//     PlcTask Inputs/GVL_iXlinker.EtherCAT_Master_EPPxxxx.Beckhoff_EPP1xxx.Beckhoff_EPP1xxxEK1122.A_0018_EPP1321_0060_0016.A_0019_EPP1322_0001_0016.A_0020_EPP1322_0001_0017.A_0021_EPP1332_0001_0016.A_0022_EPP1332_0001_0017.A_0023_EPP1342_0001_0016.A_0024_EPP1342_0001_0017.A_0027_EPP1809_0021_0016.WcState.WcState <-> WcState/WcState
//     PlcTask Inputs/GVL_iXlinker.EtherCAT_Master_EPPxxxx.Beckhoff_EPP1xxx.Beckhoff_EPP1xxxEK1122.A_0018_EPP1321_0060_0016.A_0019_EPP1322_0001_0016.A_0020_EPP1322_0001_0017.A_0021_EPP1332_0001_0016.A_0022_EPP1332_0001_0017.A_0023_EPP1342_0001_0016.A_0024_EPP1342_0001_0017.A_0027_EPP1809_0021_0016.WcState.InputToggle <-> WcState/InputToggle
//     PlcTask Inputs/GVL_iXlinker.EtherCAT_Master_EPPxxxx.Beckhoff_EPP1xxx.Beckhoff_EPP1xxxEK1122.A_0018_EPP1321_0060_0016.A_0019_EPP1322_0001_0016.A_0020_EPP1322_0001_0017.A_0021_EPP1332_0001_0016.A_0022_EPP1332_0001_0017.A_0023_EPP1342_0001_0016.A_0024_EPP1342_0001_0017.A_0027_EPP1809_0021_0016.InfoData.State <-> InfoData/State
//   PLC/PLC Instance <-> EtherCAT Master EPPxxxx/Beckhoff EPP1xxx/Beckhoff EPP1xxxEK1122/A_0018(EPP1321-0060-0016)/A_0019(EPP1322-0001-0016)/A_0020(EPP1322-0001-0017)/A_0021(EPP1332-0001-0016)/A_0022(EPP1332-0001-0017)/A_0023(EPP1342-0001-0016)/A_0024(EPP1342-0001-0017)/A_0028(EPP1809-0022-0016)
//     PlcTask Inputs/GVL_iXlinker.EtherCAT_Master_EPPxxxx.Beckhoff_EPP1xxx.Beckhoff_EPP1xxxEK1122.A_0018_EPP1321_0060_0016.A_0019_EPP1322_0001_0016.A_0020_EPP1322_0001_0017.A_0021_EPP1332_0001_0016.A_0022_EPP1332_0001_0017.A_0023_EPP1342_0001_0016.A_0024_EPP1342_0001_0017.A_0028_EPP1809_0022_0016.Channel_1.Input <-> Channel 1/Input
//     PlcTask Inputs/GVL_iXlinker.EtherCAT_Master_EPPxxxx.Beckhoff_EPP1xxx.Beckhoff_EPP1xxxEK1122.A_0018_EPP1321_0060_0016.A_0019_EPP1322_0001_0016.A_0020_EPP1322_0001_0017.A_0021_EPP1332_0001_0016.A_0022_EPP1332_0001_0017.A_0023_EPP1342_0001_0016.A_0024_EPP1342_0001_0017.A_0028_EPP1809_0022_0016.Channel_2.Input <-> Channel 2/Input
//     PlcTask Inputs/GVL_iXlinker.EtherCAT_Master_EPPxxxx.Beckhoff_EPP1xxx.Beckhoff_EPP1xxxEK1122.A_0018_EPP1321_0060_0016.A_0019_EPP1322_0001_0016.A_0020_EPP1322_0001_0017.A_0021_EPP1332_0001_0016.A_0022_EPP1332_0001_0017.A_0023_EPP1342_0001_0016.A_0024_EPP1342_0001_0017.A_0028_EPP1809_0022_0016.Channel_3.Input <-> Channel 3/Input
//     PlcTask Inputs/GVL_iXlinker.EtherCAT_Master_EPPxxxx.Beckhoff_EPP1xxx.Beckhoff_EPP1xxxEK1122.A_0018_EPP1321_0060_0016.A_0019_EPP1322_0001_0016.A_0020_EPP1322_0001_0017.A_0021_EPP1332_0001_0016.A_0022_EPP1332_0001_0017.A_0023_EPP1342_0001_0016.A_0024_EPP1342_0001_0017.A_0028_EPP1809_0022_0016.Channel_4.Input <-> Channel 4/Input
//     PlcTask Inputs/GVL_iXlinker.EtherCAT_Master_EPPxxxx.Beckhoff_EPP1xxx.Beckhoff_EPP1xxxEK1122.A_0018_EPP1321_0060_0016.A_0019_EPP1322_0001_0016.A_0020_EPP1322_0001_0017.A_0021_EPP1332_0001_0016.A_0022_EPP1332_0001_0017.A_0023_EPP1342_0001_0016.A_0024_EPP1342_0001_0017.A_0028_EPP1809_0022_0016.Channel_5.Input <-> Channel 5/Input
//     PlcTask Inputs/GVL_iXlinker.EtherCAT_Master_EPPxxxx.Beckhoff_EPP1xxx.Beckhoff_EPP1xxxEK1122.A_0018_EPP1321_0060_0016.A_0019_EPP1322_0001_0016.A_0020_EPP1322_0001_0017.A_0021_EPP1332_0001_0016.A_0022_EPP1332_0001_0017.A_0023_EPP1342_0001_0016.A_0024_EPP1342_0001_0017.A_0028_EPP1809_0022_0016.Channel_6.Input <-> Channel 6/Input
//     PlcTask Inputs/GVL_iXlinker.EtherCAT_Master_EPPxxxx.Beckhoff_EPP1xxx.Beckhoff_EPP1xxxEK1122.A_0018_EPP1321_0060_0016.A_0019_EPP1322_0001_0016.A_0020_EPP1322_0001_0017.A_0021_EPP1332_0001_0016.A_0022_EPP1332_0001_0017.A_0023_EPP1342_0001_0016.A_0024_EPP1342_0001_0017.A_0028_EPP1809_0022_0016.Channel_7.Input <-> Channel 7/Input
//     PlcTask Inputs/GVL_iXlinker.EtherCAT_Master_EPPxxxx.Beckhoff_EPP1xxx.Beckhoff_EPP1xxxEK1122.A_0018_EPP1321_0060_0016.A_0019_EPP1322_0001_0016.A_0020_EPP1322_0001_0017.A_0021_EPP1332_0001_0016.A_0022_EPP1332_0001_0017.A_0023_EPP1342_0001_0016.A_0024_EPP1342_0001_0017.A_0028_EPP1809_0022_0016.Channel_8.Input <-> Channel 8/Input
//     PlcTask Inputs/GVL_iXlinker.EtherCAT_Master_EPPxxxx.Beckhoff_EPP1xxx.Beckhoff_EPP1xxxEK1122.A_0018_EPP1321_0060_0016.A_0019_EPP1322_0001_0016.A_0020_EPP1322_0001_0017.A_0021_EPP1332_0001_0016.A_0022_EPP1332_0001_0017.A_0023_EPP1342_0001_0016.A_0024_EPP1342_0001_0017.A_0028_EPP1809_0022_0016.Channel_9.Input <-> Channel 9/Input
//     PlcTask Inputs/GVL_iXlinker.EtherCAT_Master_EPPxxxx.Beckhoff_EPP1xxx.Beckhoff_EPP1xxxEK1122.A_0018_EPP1321_0060_0016.A_0019_EPP1322_0001_0016.A_0020_EPP1322_0001_0017.A_0021_EPP1332_0001_0016.A_0022_EPP1332_0001_0017.A_0023_EPP1342_0001_0016.A_0024_EPP1342_0001_0017.A_0028_EPP1809_0022_0016.Channel_10.Input <-> Channel 10/Input
//     PlcTask Inputs/GVL_iXlinker.EtherCAT_Master_EPPxxxx.Beckhoff_EPP1xxx.Beckhoff_EPP1xxxEK1122.A_0018_EPP1321_0060_0016.A_0019_EPP1322_0001_0016.A_0020_EPP1322_0001_0017.A_0021_EPP1332_0001_0016.A_0022_EPP1332_0001_0017.A_0023_EPP1342_0001_0016.A_0024_EPP1342_0001_0017.A_0028_EPP1809_0022_0016.Channel_11.Input <-> Channel 11/Input
//     PlcTask Inputs/GVL_iXlinker.EtherCAT_Master_EPPxxxx.Beckhoff_EPP1xxx.Beckhoff_EPP1xxxEK1122.A_0018_EPP1321_0060_0016.A_0019_EPP1322_0001_0016.A_0020_EPP1322_0001_0017.A_0021_EPP1332_0001_0016.A_0022_EPP1332_0001_0017.A_0023_EPP1342_0001_0016.A_0024_EPP1342_0001_0017.A_0028_EPP1809_0022_0016.Channel_12.Input <-> Channel 12/Input
//     PlcTask Inputs/GVL_iXlinker.EtherCAT_Master_EPPxxxx.Beckhoff_EPP1xxx.Beckhoff_EPP1xxxEK1122.A_0018_EPP1321_0060_0016.A_0019_EPP1322_0001_0016.A_0020_EPP1322_0001_0017.A_0021_EPP1332_0001_0016.A_0022_EPP1332_0001_0017.A_0023_EPP1342_0001_0016.A_0024_EPP1342_0001_0017.A_0028_EPP1809_0022_0016.Channel_13.Input <-> Channel 13/Input
//     PlcTask Inputs/GVL_iXlinker.EtherCAT_Master_EPPxxxx.Beckhoff_EPP1xxx.Beckhoff_EPP1xxxEK1122.A_0018_EPP1321_0060_0016.A_0019_EPP1322_0001_0016.A_0020_EPP1322_0001_0017.A_0021_EPP1332_0001_0016.A_0022_EPP1332_0001_0017.A_0023_EPP1342_0001_0016.A_0024_EPP1342_0001_0017.A_0028_EPP1809_0022_0016.Channel_14.Input <-> Channel 14/Input
//     PlcTask Inputs/GVL_iXlinker.EtherCAT_Master_EPPxxxx.Beckhoff_EPP1xxx.Beckhoff_EPP1xxxEK1122.A_0018_EPP1321_0060_0016.A_0019_EPP1322_0001_0016.A_0020_EPP1322_0001_0017.A_0021_EPP1332_0001_0016.A_0022_EPP1332_0001_0017.A_0023_EPP1342_0001_0016.A_0024_EPP1342_0001_0017.A_0028_EPP1809_0022_0016.Channel_15.Input <-> Channel 15/Input
//     PlcTask Inputs/GVL_iXlinker.EtherCAT_Master_EPPxxxx.Beckhoff_EPP1xxx.Beckhoff_EPP1xxxEK1122.A_0018_EPP1321_0060_0016.A_0019_EPP1322_0001_0016.A_0020_EPP1322_0001_0017.A_0021_EPP1332_0001_0016.A_0022_EPP1332_0001_0017.A_0023_EPP1342_0001_0016.A_0024_EPP1342_0001_0017.A_0028_EPP1809_0022_0016.Channel_16.Input <-> Channel 16/Input
//     PlcTask Inputs/GVL_iXlinker.EtherCAT_Master_EPPxxxx.Beckhoff_EPP1xxx.Beckhoff_EPP1xxxEK1122.A_0018_EPP1321_0060_0016.A_0019_EPP1322_0001_0016.A_0020_EPP1322_0001_0017.A_0021_EPP1332_0001_0016.A_0022_EPP1332_0001_0017.A_0023_EPP1342_0001_0016.A_0024_EPP1342_0001_0017.A_0028_EPP1809_0022_0016.WcState.WcState <-> WcState/WcState
//     PlcTask Inputs/GVL_iXlinker.EtherCAT_Master_EPPxxxx.Beckhoff_EPP1xxx.Beckhoff_EPP1xxxEK1122.A_0018_EPP1321_0060_0016.A_0019_EPP1322_0001_0016.A_0020_EPP1322_0001_0017.A_0021_EPP1332_0001_0016.A_0022_EPP1332_0001_0017.A_0023_EPP1342_0001_0016.A_0024_EPP1342_0001_0017.A_0028_EPP1809_0022_0016.WcState.InputToggle <-> WcState/InputToggle
//     PlcTask Inputs/GVL_iXlinker.EtherCAT_Master_EPPxxxx.Beckhoff_EPP1xxx.Beckhoff_EPP1xxxEK1122.A_0018_EPP1321_0060_0016.A_0019_EPP1322_0001_0016.A_0020_EPP1322_0001_0017.A_0021_EPP1332_0001_0016.A_0022_EPP1332_0001_0017.A_0023_EPP1342_0001_0016.A_0024_EPP1342_0001_0017.A_0028_EPP1809_0022_0016.InfoData.State <-> InfoData/State
//   PLC/PLC Instance <-> EtherCAT Master EPPxxxx/Beckhoff EPP1xxx/Beckhoff EPP1xxxEK1122/A_0018(EPP1321-0060-0016)/A_0019(EPP1322-0001-0016)/A_0020(EPP1322-0001-0017)/A_0021(EPP1332-0001-0016)/A_0022(EPP1332-0001-0017)/A_0023(EPP1342-0001-0016)/A_0024(EPP1342-0001-0017)/A_0029(EPP1819-0021-0016)
//     PlcTask Inputs/GVL_iXlinker.EtherCAT_Master_EPPxxxx.Beckhoff_EPP1xxx.Beckhoff_EPP1xxxEK1122.A_0018_EPP1321_0060_0016.A_0019_EPP1322_0001_0016.A_0020_EPP1322_0001_0017.A_0021_EPP1332_0001_0016.A_0022_EPP1332_0001_0017.A_0023_EPP1342_0001_0016.A_0024_EPP1342_0001_0017.A_0029_EPP1819_0021_0016.Channel_1.Input <-> Channel 1/Input
//     PlcTask Inputs/GVL_iXlinker.EtherCAT_Master_EPPxxxx.Beckhoff_EPP1xxx.Beckhoff_EPP1xxxEK1122.A_0018_EPP1321_0060_0016.A_0019_EPP1322_0001_0016.A_0020_EPP1322_0001_0017.A_0021_EPP1332_0001_0016.A_0022_EPP1332_0001_0017.A_0023_EPP1342_0001_0016.A_0024_EPP1342_0001_0017.A_0029_EPP1819_0021_0016.Channel_2.Input <-> Channel 2/Input
//     PlcTask Inputs/GVL_iXlinker.EtherCAT_Master_EPPxxxx.Beckhoff_EPP1xxx.Beckhoff_EPP1xxxEK1122.A_0018_EPP1321_0060_0016.A_0019_EPP1322_0001_0016.A_0020_EPP1322_0001_0017.A_0021_EPP1332_0001_0016.A_0022_EPP1332_0001_0017.A_0023_EPP1342_0001_0016.A_0024_EPP1342_0001_0017.A_0029_EPP1819_0021_0016.Channel_3.Input <-> Channel 3/Input
//     PlcTask Inputs/GVL_iXlinker.EtherCAT_Master_EPPxxxx.Beckhoff_EPP1xxx.Beckhoff_EPP1xxxEK1122.A_0018_EPP1321_0060_0016.A_0019_EPP1322_0001_0016.A_0020_EPP1322_0001_0017.A_0021_EPP1332_0001_0016.A_0022_EPP1332_0001_0017.A_0023_EPP1342_0001_0016.A_0024_EPP1342_0001_0017.A_0029_EPP1819_0021_0016.Channel_4.Input <-> Channel 4/Input
//     PlcTask Inputs/GVL_iXlinker.EtherCAT_Master_EPPxxxx.Beckhoff_EPP1xxx.Beckhoff_EPP1xxxEK1122.A_0018_EPP1321_0060_0016.A_0019_EPP1322_0001_0016.A_0020_EPP1322_0001_0017.A_0021_EPP1332_0001_0016.A_0022_EPP1332_0001_0017.A_0023_EPP1342_0001_0016.A_0024_EPP1342_0001_0017.A_0029_EPP1819_0021_0016.Channel_5.Input <-> Channel 5/Input
//     PlcTask Inputs/GVL_iXlinker.EtherCAT_Master_EPPxxxx.Beckhoff_EPP1xxx.Beckhoff_EPP1xxxEK1122.A_0018_EPP1321_0060_0016.A_0019_EPP1322_0001_0016.A_0020_EPP1322_0001_0017.A_0021_EPP1332_0001_0016.A_0022_EPP1332_0001_0017.A_0023_EPP1342_0001_0016.A_0024_EPP1342_0001_0017.A_0029_EPP1819_0021_0016.Channel_6.Input <-> Channel 6/Input
//     PlcTask Inputs/GVL_iXlinker.EtherCAT_Master_EPPxxxx.Beckhoff_EPP1xxx.Beckhoff_EPP1xxxEK1122.A_0018_EPP1321_0060_0016.A_0019_EPP1322_0001_0016.A_0020_EPP1322_0001_0017.A_0021_EPP1332_0001_0016.A_0022_EPP1332_0001_0017.A_0023_EPP1342_0001_0016.A_0024_EPP1342_0001_0017.A_0029_EPP1819_0021_0016.Channel_7.Input <-> Channel 7/Input
//     PlcTask Inputs/GVL_iXlinker.EtherCAT_Master_EPPxxxx.Beckhoff_EPP1xxx.Beckhoff_EPP1xxxEK1122.A_0018_EPP1321_0060_0016.A_0019_EPP1322_0001_0016.A_0020_EPP1322_0001_0017.A_0021_EPP1332_0001_0016.A_0022_EPP1332_0001_0017.A_0023_EPP1342_0001_0016.A_0024_EPP1342_0001_0017.A_0029_EPP1819_0021_0016.Channel_8.Input <-> Channel 8/Input
//     PlcTask Inputs/GVL_iXlinker.EtherCAT_Master_EPPxxxx.Beckhoff_EPP1xxx.Beckhoff_EPP1xxxEK1122.A_0018_EPP1321_0060_0016.A_0019_EPP1322_0001_0016.A_0020_EPP1322_0001_0017.A_0021_EPP1332_0001_0016.A_0022_EPP1332_0001_0017.A_0023_EPP1342_0001_0016.A_0024_EPP1342_0001_0017.A_0029_EPP1819_0021_0016.Channel_9.Input <-> Channel 9/Input
//     PlcTask Inputs/GVL_iXlinker.EtherCAT_Master_EPPxxxx.Beckhoff_EPP1xxx.Beckhoff_EPP1xxxEK1122.A_0018_EPP1321_0060_0016.A_0019_EPP1322_0001_0016.A_0020_EPP1322_0001_0017.A_0021_EPP1332_0001_0016.A_0022_EPP1332_0001_0017.A_0023_EPP1342_0001_0016.A_0024_EPP1342_0001_0017.A_0029_EPP1819_0021_0016.Channel_10.Input <-> Channel 10/Input
//     PlcTask Inputs/GVL_iXlinker.EtherCAT_Master_EPPxxxx.Beckhoff_EPP1xxx.Beckhoff_EPP1xxxEK1122.A_0018_EPP1321_0060_0016.A_0019_EPP1322_0001_0016.A_0020_EPP1322_0001_0017.A_0021_EPP1332_0001_0016.A_0022_EPP1332_0001_0017.A_0023_EPP1342_0001_0016.A_0024_EPP1342_0001_0017.A_0029_EPP1819_0021_0016.Channel_11.Input <-> Channel 11/Input
//     PlcTask Inputs/GVL_iXlinker.EtherCAT_Master_EPPxxxx.Beckhoff_EPP1xxx.Beckhoff_EPP1xxxEK1122.A_0018_EPP1321_0060_0016.A_0019_EPP1322_0001_0016.A_0020_EPP1322_0001_0017.A_0021_EPP1332_0001_0016.A_0022_EPP1332_0001_0017.A_0023_EPP1342_0001_0016.A_0024_EPP1342_0001_0017.A_0029_EPP1819_0021_0016.Channel_12.Input <-> Channel 12/Input
//     PlcTask Inputs/GVL_iXlinker.EtherCAT_Master_EPPxxxx.Beckhoff_EPP1xxx.Beckhoff_EPP1xxxEK1122.A_0018_EPP1321_0060_0016.A_0019_EPP1322_0001_0016.A_0020_EPP1322_0001_0017.A_0021_EPP1332_0001_0016.A_0022_EPP1332_0001_0017.A_0023_EPP1342_0001_0016.A_0024_EPP1342_0001_0017.A_0029_EPP1819_0021_0016.Channel_13.Input <-> Channel 13/Input
//     PlcTask Inputs/GVL_iXlinker.EtherCAT_Master_EPPxxxx.Beckhoff_EPP1xxx.Beckhoff_EPP1xxxEK1122.A_0018_EPP1321_0060_0016.A_0019_EPP1322_0001_0016.A_0020_EPP1322_0001_0017.A_0021_EPP1332_0001_0016.A_0022_EPP1332_0001_0017.A_0023_EPP1342_0001_0016.A_0024_EPP1342_0001_0017.A_0029_EPP1819_0021_0016.Channel_14.Input <-> Channel 14/Input
//     PlcTask Inputs/GVL_iXlinker.EtherCAT_Master_EPPxxxx.Beckhoff_EPP1xxx.Beckhoff_EPP1xxxEK1122.A_0018_EPP1321_0060_0016.A_0019_EPP1322_0001_0016.A_0020_EPP1322_0001_0017.A_0021_EPP1332_0001_0016.A_0022_EPP1332_0001_0017.A_0023_EPP1342_0001_0016.A_0024_EPP1342_0001_0017.A_0029_EPP1819_0021_0016.Channel_15.Input <-> Channel 15/Input
//     PlcTask Inputs/GVL_iXlinker.EtherCAT_Master_EPPxxxx.Beckhoff_EPP1xxx.Beckhoff_EPP1xxxEK1122.A_0018_EPP1321_0060_0016.A_0019_EPP1322_0001_0016.A_0020_EPP1322_0001_0017.A_0021_EPP1332_0001_0016.A_0022_EPP1332_0001_0017.A_0023_EPP1342_0001_0016.A_0024_EPP1342_0001_0017.A_0029_EPP1819_0021_0016.Channel_16.Input <-> Channel 16/Input
//     PlcTask Inputs/GVL_iXlinker.EtherCAT_Master_EPPxxxx.Beckhoff_EPP1xxx.Beckhoff_EPP1xxxEK1122.A_0018_EPP1321_0060_0016.A_0019_EPP1322_0001_0016.A_0020_EPP1322_0001_0017.A_0021_EPP1332_0001_0016.A_0022_EPP1332_0001_0017.A_0023_EPP1342_0001_0016.A_0024_EPP1342_0001_0017.A_0029_EPP1819_0021_0016.WcState.WcState <-> WcState/WcState
//     PlcTask Inputs/GVL_iXlinker.EtherCAT_Master_EPPxxxx.Beckhoff_EPP1xxx.Beckhoff_EPP1xxxEK1122.A_0018_EPP1321_0060_0016.A_0019_EPP1322_0001_0016.A_0020_EPP1322_0001_0017.A_0021_EPP1332_0001_0016.A_0022_EPP1332_0001_0017.A_0023_EPP1342_0001_0016.A_0024_EPP1342_0001_0017.A_0029_EPP1819_0021_0016.WcState.InputToggle <-> WcState/InputToggle
//     PlcTask Inputs/GVL_iXlinker.EtherCAT_Master_EPPxxxx.Beckhoff_EPP1xxx.Beckhoff_EPP1xxxEK1122.A_0018_EPP1321_0060_0016.A_0019_EPP1322_0001_0016.A_0020_EPP1322_0001_0017.A_0021_EPP1332_0001_0016.A_0022_EPP1332_0001_0017.A_0023_EPP1342_0001_0016.A_0024_EPP1342_0001_0017.A_0029_EPP1819_0021_0016.InfoData.State <-> InfoData/State
//   PLC/PLC Instance <-> EtherCAT Master EPPxxxx/Beckhoff EPP1xxx/Beckhoff EPP1xxxEK1122/A_0018(EPP1321-0060-0016)/A_0019(EPP1322-0001-0016)/A_0020(EPP1322-0001-0017)/A_0021(EPP1332-0001-0016)/A_0022(EPP1332-0001-0017)/A_0023(EPP1342-0001-0016)/A_0024(EPP1342-0001-0017)/A_0030(EPP1819-0022-0016)
//     PlcTask Inputs/GVL_iXlinker.EtherCAT_Master_EPPxxxx.Beckhoff_EPP1xxx.Beckhoff_EPP1xxxEK1122.A_0018_EPP1321_0060_0016.A_0019_EPP1322_0001_0016.A_0020_EPP1322_0001_0017.A_0021_EPP1332_0001_0016.A_0022_EPP1332_0001_0017.A_0023_EPP1342_0001_0016.A_0024_EPP1342_0001_0017.A_0030_EPP1819_0022_0016.Channel_1.Input <-> Channel 1/Input
//     PlcTask Inputs/GVL_iXlinker.EtherCAT_Master_EPPxxxx.Beckhoff_EPP1xxx.Beckhoff_EPP1xxxEK1122.A_0018_EPP1321_0060_0016.A_0019_EPP1322_0001_0016.A_0020_EPP1322_0001_0017.A_0021_EPP1332_0001_0016.A_0022_EPP1332_0001_0017.A_0023_EPP1342_0001_0016.A_0024_EPP1342_0001_0017.A_0030_EPP1819_0022_0016.Channel_2.Input <-> Channel 2/Input
//     PlcTask Inputs/GVL_iXlinker.EtherCAT_Master_EPPxxxx.Beckhoff_EPP1xxx.Beckhoff_EPP1xxxEK1122.A_0018_EPP1321_0060_0016.A_0019_EPP1322_0001_0016.A_0020_EPP1322_0001_0017.A_0021_EPP1332_0001_0016.A_0022_EPP1332_0001_0017.A_0023_EPP1342_0001_0016.A_0024_EPP1342_0001_0017.A_0030_EPP1819_0022_0016.Channel_3.Input <-> Channel 3/Input
//     PlcTask Inputs/GVL_iXlinker.EtherCAT_Master_EPPxxxx.Beckhoff_EPP1xxx.Beckhoff_EPP1xxxEK1122.A_0018_EPP1321_0060_0016.A_0019_EPP1322_0001_0016.A_0020_EPP1322_0001_0017.A_0021_EPP1332_0001_0016.A_0022_EPP1332_0001_0017.A_0023_EPP1342_0001_0016.A_0024_EPP1342_0001_0017.A_0030_EPP1819_0022_0016.Channel_4.Input <-> Channel 4/Input
//     PlcTask Inputs/GVL_iXlinker.EtherCAT_Master_EPPxxxx.Beckhoff_EPP1xxx.Beckhoff_EPP1xxxEK1122.A_0018_EPP1321_0060_0016.A_0019_EPP1322_0001_0016.A_0020_EPP1322_0001_0017.A_0021_EPP1332_0001_0016.A_0022_EPP1332_0001_0017.A_0023_EPP1342_0001_0016.A_0024_EPP1342_0001_0017.A_0030_EPP1819_0022_0016.Channel_5.Input <-> Channel 5/Input
//     PlcTask Inputs/GVL_iXlinker.EtherCAT_Master_EPPxxxx.Beckhoff_EPP1xxx.Beckhoff_EPP1xxxEK1122.A_0018_EPP1321_0060_0016.A_0019_EPP1322_0001_0016.A_0020_EPP1322_0001_0017.A_0021_EPP1332_0001_0016.A_0022_EPP1332_0001_0017.A_0023_EPP1342_0001_0016.A_0024_EPP1342_0001_0017.A_0030_EPP1819_0022_0016.Channel_6.Input <-> Channel 6/Input
//     PlcTask Inputs/GVL_iXlinker.EtherCAT_Master_EPPxxxx.Beckhoff_EPP1xxx.Beckhoff_EPP1xxxEK1122.A_0018_EPP1321_0060_0016.A_0019_EPP1322_0001_0016.A_0020_EPP1322_0001_0017.A_0021_EPP1332_0001_0016.A_0022_EPP1332_0001_0017.A_0023_EPP1342_0001_0016.A_0024_EPP1342_0001_0017.A_0030_EPP1819_0022_0016.Channel_7.Input <-> Channel 7/Input
//     PlcTask Inputs/GVL_iXlinker.EtherCAT_Master_EPPxxxx.Beckhoff_EPP1xxx.Beckhoff_EPP1xxxEK1122.A_0018_EPP1321_0060_0016.A_0019_EPP1322_0001_0016.A_0020_EPP1322_0001_0017.A_0021_EPP1332_0001_0016.A_0022_EPP1332_0001_0017.A_0023_EPP1342_0001_0016.A_0024_EPP1342_0001_0017.A_0030_EPP1819_0022_0016.Channel_8.Input <-> Channel 8/Input
//     PlcTask Inputs/GVL_iXlinker.EtherCAT_Master_EPPxxxx.Beckhoff_EPP1xxx.Beckhoff_EPP1xxxEK1122.A_0018_EPP1321_0060_0016.A_0019_EPP1322_0001_0016.A_0020_EPP1322_0001_0017.A_0021_EPP1332_0001_0016.A_0022_EPP1332_0001_0017.A_0023_EPP1342_0001_0016.A_0024_EPP1342_0001_0017.A_0030_EPP1819_0022_0016.Channel_9.Input <-> Channel 9/Input
//     PlcTask Inputs/GVL_iXlinker.EtherCAT_Master_EPPxxxx.Beckhoff_EPP1xxx.Beckhoff_EPP1xxxEK1122.A_0018_EPP1321_0060_0016.A_0019_EPP1322_0001_0016.A_0020_EPP1322_0001_0017.A_0021_EPP1332_0001_0016.A_0022_EPP1332_0001_0017.A_0023_EPP1342_0001_0016.A_0024_EPP1342_0001_0017.A_0030_EPP1819_0022_0016.Channel_10.Input <-> Channel 10/Input
//     PlcTask Inputs/GVL_iXlinker.EtherCAT_Master_EPPxxxx.Beckhoff_EPP1xxx.Beckhoff_EPP1xxxEK1122.A_0018_EPP1321_0060_0016.A_0019_EPP1322_0001_0016.A_0020_EPP1322_0001_0017.A_0021_EPP1332_0001_0016.A_0022_EPP1332_0001_0017.A_0023_EPP1342_0001_0016.A_0024_EPP1342_0001_0017.A_0030_EPP1819_0022_0016.Channel_11.Input <-> Channel 11/Input
//     PlcTask Inputs/GVL_iXlinker.EtherCAT_Master_EPPxxxx.Beckhoff_EPP1xxx.Beckhoff_EPP1xxxEK1122.A_0018_EPP1321_0060_0016.A_0019_EPP1322_0001_0016.A_0020_EPP1322_0001_0017.A_0021_EPP1332_0001_0016.A_0022_EPP1332_0001_0017.A_0023_EPP1342_0001_0016.A_0024_EPP1342_0001_0017.A_0030_EPP1819_0022_0016.Channel_12.Input <-> Channel 12/Input
//     PlcTask Inputs/GVL_iXlinker.EtherCAT_Master_EPPxxxx.Beckhoff_EPP1xxx.Beckhoff_EPP1xxxEK1122.A_0018_EPP1321_0060_0016.A_0019_EPP1322_0001_0016.A_0020_EPP1322_0001_0017.A_0021_EPP1332_0001_0016.A_0022_EPP1332_0001_0017.A_0023_EPP1342_0001_0016.A_0024_EPP1342_0001_0017.A_0030_EPP1819_0022_0016.Channel_13.Input <-> Channel 13/Input
//     PlcTask Inputs/GVL_iXlinker.EtherCAT_Master_EPPxxxx.Beckhoff_EPP1xxx.Beckhoff_EPP1xxxEK1122.A_0018_EPP1321_0060_0016.A_0019_EPP1322_0001_0016.A_0020_EPP1322_0001_0017.A_0021_EPP1332_0001_0016.A_0022_EPP1332_0001_0017.A_0023_EPP1342_0001_0016.A_0024_EPP1342_0001_0017.A_0030_EPP1819_0022_0016.Channel_14.Input <-> Channel 14/Input
//     PlcTask Inputs/GVL_iXlinker.EtherCAT_Master_EPPxxxx.Beckhoff_EPP1xxx.Beckhoff_EPP1xxxEK1122.A_0018_EPP1321_0060_0016.A_0019_EPP1322_0001_0016.A_0020_EPP1322_0001_0017.A_0021_EPP1332_0001_0016.A_0022_EPP1332_0001_0017.A_0023_EPP1342_0001_0016.A_0024_EPP1342_0001_0017.A_0030_EPP1819_0022_0016.Channel_15.Input <-> Channel 15/Input
//     PlcTask Inputs/GVL_iXlinker.EtherCAT_Master_EPPxxxx.Beckhoff_EPP1xxx.Beckhoff_EPP1xxxEK1122.A_0018_EPP1321_0060_0016.A_0019_EPP1322_0001_0016.A_0020_EPP1322_0001_0017.A_0021_EPP1332_0001_0016.A_0022_EPP1332_0001_0017.A_0023_EPP1342_0001_0016.A_0024_EPP1342_0001_0017.A_0030_EPP1819_0022_0016.Channel_16.Input <-> Channel 16/Input
//     PlcTask Inputs/GVL_iXlinker.EtherCAT_Master_EPPxxxx.Beckhoff_EPP1xxx.Beckhoff_EPP1xxxEK1122.A_0018_EPP1321_0060_0016.A_0019_EPP1322_0001_0016.A_0020_EPP1322_0001_0017.A_0021_EPP1332_0001_0016.A_0022_EPP1332_0001_0017.A_0023_EPP1342_0001_0016.A_0024_EPP1342_0001_0017.A_0030_EPP1819_0022_0016.WcState.WcState <-> WcState/WcState
//     PlcTask Inputs/GVL_iXlinker.EtherCAT_Master_EPPxxxx.Beckhoff_EPP1xxx.Beckhoff_EPP1xxxEK1122.A_0018_EPP1321_0060_0016.A_0019_EPP1322_0001_0016.A_0020_EPP1322_0001_0017.A_0021_EPP1332_0001_0016.A_0022_EPP1332_0001_0017.A_0023_EPP1342_0001_0016.A_0024_EPP1342_0001_0017.A_0030_EPP1819_0022_0016.WcState.InputToggle <-> WcState/InputToggle
//     PlcTask Inputs/GVL_iXlinker.EtherCAT_Master_EPPxxxx.Beckhoff_EPP1xxx.Beckhoff_EPP1xxxEK1122.A_0018_EPP1321_0060_0016.A_0019_EPP1322_0001_0016.A_0020_EPP1322_0001_0017.A_0021_EPP1332_0001_0016.A_0022_EPP1332_0001_0017.A_0023_EPP1342_0001_0016.A_0024_EPP1342_0001_0017.A_0030_EPP1819_0022_0016.InfoData.State <-> InfoData/State
//   PLC/PLC Instance <-> EtherCAT Master EPPxxxx/Beckhoff EPP1xxx/Beckhoff EPP1xxxEK1122/A_0018(EPP1321-0060-0016)/A_0019(EPP1322-0001-0016)/A_0020(EPP1322-0001-0017)/A_0021(EPP1332-0001-0016)/A_0022(EPP1332-0001-0017)/A_0023(EPP1342-0001-0016)/A_0024(EPP1342-0001-0017)/A_0031(EPP1816-0003-0016)
//     PlcTask Inputs/GVL_iXlinker.EtherCAT_Master_EPPxxxx.Beckhoff_EPP1xxx.Beckhoff_EPP1xxxEK1122.A_0018_EPP1321_0060_0016.A_0019_EPP1322_0001_0016.A_0020_EPP1322_0001_0017.A_0021_EPP1332_0001_0016.A_0022_EPP1332_0001_0017.A_0023_EPP1342_0001_0016.A_0024_EPP1342_0001_0017.A_0031_EPP1816_0003_0016.DIG_Inputs_Channel_1.Input[0] <-> DIG Inputs Channel 1/Input 1
//     PlcTask Inputs/GVL_iXlinker.EtherCAT_Master_EPPxxxx.Beckhoff_EPP1xxx.Beckhoff_EPP1xxxEK1122.A_0018_EPP1321_0060_0016.A_0019_EPP1322_0001_0016.A_0020_EPP1322_0001_0017.A_0021_EPP1332_0001_0016.A_0022_EPP1332_0001_0017.A_0023_EPP1342_0001_0016.A_0024_EPP1342_0001_0017.A_0031_EPP1816_0003_0016.DIG_Inputs_Channel_1.Input[1] <-> DIG Inputs Channel 1/Input 2
//     PlcTask Inputs/GVL_iXlinker.EtherCAT_Master_EPPxxxx.Beckhoff_EPP1xxx.Beckhoff_EPP1xxxEK1122.A_0018_EPP1321_0060_0016.A_0019_EPP1322_0001_0016.A_0020_EPP1322_0001_0017.A_0021_EPP1332_0001_0016.A_0022_EPP1332_0001_0017.A_0023_EPP1342_0001_0016.A_0024_EPP1342_0001_0017.A_0031_EPP1816_0003_0016.DIG_Inputs_Channel_1.Input[2] <-> DIG Inputs Channel 1/Input 3
//     PlcTask Inputs/GVL_iXlinker.EtherCAT_Master_EPPxxxx.Beckhoff_EPP1xxx.Beckhoff_EPP1xxxEK1122.A_0018_EPP1321_0060_0016.A_0019_EPP1322_0001_0016.A_0020_EPP1322_0001_0017.A_0021_EPP1332_0001_0016.A_0022_EPP1332_0001_0017.A_0023_EPP1342_0001_0016.A_0024_EPP1342_0001_0017.A_0031_EPP1816_0003_0016.DIG_Inputs_Channel_1.Input[3] <-> DIG Inputs Channel 1/Input 4
//     PlcTask Inputs/GVL_iXlinker.EtherCAT_Master_EPPxxxx.Beckhoff_EPP1xxx.Beckhoff_EPP1xxxEK1122.A_0018_EPP1321_0060_0016.A_0019_EPP1322_0001_0016.A_0020_EPP1322_0001_0017.A_0021_EPP1332_0001_0016.A_0022_EPP1332_0001_0017.A_0023_EPP1342_0001_0016.A_0024_EPP1342_0001_0017.A_0031_EPP1816_0003_0016.DIG_Inputs_Channel_1.Input[4] <-> DIG Inputs Channel 1/Input 5
//     PlcTask Inputs/GVL_iXlinker.EtherCAT_Master_EPPxxxx.Beckhoff_EPP1xxx.Beckhoff_EPP1xxxEK1122.A_0018_EPP1321_0060_0016.A_0019_EPP1322_0001_0016.A_0020_EPP1322_0001_0017.A_0021_EPP1332_0001_0016.A_0022_EPP1332_0001_0017.A_0023_EPP1342_0001_0016.A_0024_EPP1342_0001_0017.A_0031_EPP1816_0003_0016.DIG_Inputs_Channel_1.Input[5] <-> DIG Inputs Channel 1/Input 6
//     PlcTask Inputs/GVL_iXlinker.EtherCAT_Master_EPPxxxx.Beckhoff_EPP1xxx.Beckhoff_EPP1xxxEK1122.A_0018_EPP1321_0060_0016.A_0019_EPP1322_0001_0016.A_0020_EPP1322_0001_0017.A_0021_EPP1332_0001_0016.A_0022_EPP1332_0001_0017.A_0023_EPP1342_0001_0016.A_0024_EPP1342_0001_0017.A_0031_EPP1816_0003_0016.DIG_Inputs_Channel_1.Input[6] <-> DIG Inputs Channel 1/Input 7
//     PlcTask Inputs/GVL_iXlinker.EtherCAT_Master_EPPxxxx.Beckhoff_EPP1xxx.Beckhoff_EPP1xxxEK1122.A_0018_EPP1321_0060_0016.A_0019_EPP1322_0001_0016.A_0020_EPP1322_0001_0017.A_0021_EPP1332_0001_0016.A_0022_EPP1332_0001_0017.A_0023_EPP1342_0001_0016.A_0024_EPP1342_0001_0017.A_0031_EPP1816_0003_0016.DIG_Inputs_Channel_1.Input[7] <-> DIG Inputs Channel 1/Input 8
//     PlcTask Inputs/GVL_iXlinker.EtherCAT_Master_EPPxxxx.Beckhoff_EPP1xxx.Beckhoff_EPP1xxxEK1122.A_0018_EPP1321_0060_0016.A_0019_EPP1322_0001_0016.A_0020_EPP1322_0001_0017.A_0021_EPP1332_0001_0016.A_0022_EPP1332_0001_0017.A_0023_EPP1342_0001_0016.A_0024_EPP1342_0001_0017.A_0031_EPP1816_0003_0016.DIG_Inputs_Channel_2.Input[0] <-> DIG Inputs Channel 2/Input 1
//     PlcTask Inputs/GVL_iXlinker.EtherCAT_Master_EPPxxxx.Beckhoff_EPP1xxx.Beckhoff_EPP1xxxEK1122.A_0018_EPP1321_0060_0016.A_0019_EPP1322_0001_0016.A_0020_EPP1322_0001_0017.A_0021_EPP1332_0001_0016.A_0022_EPP1332_0001_0017.A_0023_EPP1342_0001_0016.A_0024_EPP1342_0001_0017.A_0031_EPP1816_0003_0016.DIG_Inputs_Channel_2.Input[1] <-> DIG Inputs Channel 2/Input 2
//     PlcTask Inputs/GVL_iXlinker.EtherCAT_Master_EPPxxxx.Beckhoff_EPP1xxx.Beckhoff_EPP1xxxEK1122.A_0018_EPP1321_0060_0016.A_0019_EPP1322_0001_0016.A_0020_EPP1322_0001_0017.A_0021_EPP1332_0001_0016.A_0022_EPP1332_0001_0017.A_0023_EPP1342_0001_0016.A_0024_EPP1342_0001_0017.A_0031_EPP1816_0003_0016.DIG_Inputs_Channel_2.Input[2] <-> DIG Inputs Channel 2/Input 3
//     PlcTask Inputs/GVL_iXlinker.EtherCAT_Master_EPPxxxx.Beckhoff_EPP1xxx.Beckhoff_EPP1xxxEK1122.A_0018_EPP1321_0060_0016.A_0019_EPP1322_0001_0016.A_0020_EPP1322_0001_0017.A_0021_EPP1332_0001_0016.A_0022_EPP1332_0001_0017.A_0023_EPP1342_0001_0016.A_0024_EPP1342_0001_0017.A_0031_EPP1816_0003_0016.DIG_Inputs_Channel_2.Input[3] <-> DIG Inputs Channel 2/Input 4
//     PlcTask Inputs/GVL_iXlinker.EtherCAT_Master_EPPxxxx.Beckhoff_EPP1xxx.Beckhoff_EPP1xxxEK1122.A_0018_EPP1321_0060_0016.A_0019_EPP1322_0001_0016.A_0020_EPP1322_0001_0017.A_0021_EPP1332_0001_0016.A_0022_EPP1332_0001_0017.A_0023_EPP1342_0001_0016.A_0024_EPP1342_0001_0017.A_0031_EPP1816_0003_0016.DIG_Inputs_Channel_2.Input[4] <-> DIG Inputs Channel 2/Input 5
//     PlcTask Inputs/GVL_iXlinker.EtherCAT_Master_EPPxxxx.Beckhoff_EPP1xxx.Beckhoff_EPP1xxxEK1122.A_0018_EPP1321_0060_0016.A_0019_EPP1322_0001_0016.A_0020_EPP1322_0001_0017.A_0021_EPP1332_0001_0016.A_0022_EPP1332_0001_0017.A_0023_EPP1342_0001_0016.A_0024_EPP1342_0001_0017.A_0031_EPP1816_0003_0016.DIG_Inputs_Channel_2.Input[5] <-> DIG Inputs Channel 2/Input 6
//     PlcTask Inputs/GVL_iXlinker.EtherCAT_Master_EPPxxxx.Beckhoff_EPP1xxx.Beckhoff_EPP1xxxEK1122.A_0018_EPP1321_0060_0016.A_0019_EPP1322_0001_0016.A_0020_EPP1322_0001_0017.A_0021_EPP1332_0001_0016.A_0022_EPP1332_0001_0017.A_0023_EPP1342_0001_0016.A_0024_EPP1342_0001_0017.A_0031_EPP1816_0003_0016.DIG_Inputs_Channel_2.Input[6] <-> DIG Inputs Channel 2/Input 7
//     PlcTask Inputs/GVL_iXlinker.EtherCAT_Master_EPPxxxx.Beckhoff_EPP1xxx.Beckhoff_EPP1xxxEK1122.A_0018_EPP1321_0060_0016.A_0019_EPP1322_0001_0016.A_0020_EPP1322_0001_0017.A_0021_EPP1332_0001_0016.A_0022_EPP1332_0001_0017.A_0023_EPP1342_0001_0016.A_0024_EPP1342_0001_0017.A_0031_EPP1816_0003_0016.DIG_Inputs_Channel_2.Input[7] <-> DIG Inputs Channel 2/Input 8
//     PlcTask Inputs/GVL_iXlinker.EtherCAT_Master_EPPxxxx.Beckhoff_EPP1xxx.Beckhoff_EPP1xxxEK1122.A_0018_EPP1321_0060_0016.A_0019_EPP1322_0001_0016.A_0020_EPP1322_0001_0017.A_0021_EPP1332_0001_0016.A_0022_EPP1332_0001_0017.A_0023_EPP1342_0001_0016.A_0024_EPP1342_0001_0017.A_0031_EPP1816_0003_0016.DIG_Inputs_Channel_1.Sync_error <-> DIG Inputs Channel 1/Sync error
//     PlcTask Inputs/GVL_iXlinker.EtherCAT_Master_EPPxxxx.Beckhoff_EPP1xxx.Beckhoff_EPP1xxxEK1122.A_0018_EPP1321_0060_0016.A_0019_EPP1322_0001_0016.A_0020_EPP1322_0001_0017.A_0021_EPP1332_0001_0016.A_0022_EPP1332_0001_0017.A_0023_EPP1342_0001_0016.A_0024_EPP1342_0001_0017.A_0031_EPP1816_0003_0016.DIG_Inputs_Channel_2.Sync_error <-> DIG Inputs Channel 2/Sync error
//     PlcTask Inputs/GVL_iXlinker.EtherCAT_Master_EPPxxxx.Beckhoff_EPP1xxx.Beckhoff_EPP1xxxEK1122.A_0018_EPP1321_0060_0016.A_0019_EPP1322_0001_0016.A_0020_EPP1322_0001_0017.A_0021_EPP1332_0001_0016.A_0022_EPP1332_0001_0017.A_0023_EPP1342_0001_0016.A_0024_EPP1342_0001_0017.A_0031_EPP1816_0003_0016.DIG_Inputs_Channel_1.TxPDO_Toggle <-> DIG Inputs Channel 1/TxPDO Toggle
//     PlcTask Inputs/GVL_iXlinker.EtherCAT_Master_EPPxxxx.Beckhoff_EPP1xxx.Beckhoff_EPP1xxxEK1122.A_0018_EPP1321_0060_0016.A_0019_EPP1322_0001_0016.A_0020_EPP1322_0001_0017.A_0021_EPP1332_0001_0016.A_0022_EPP1332_0001_0017.A_0023_EPP1342_0001_0016.A_0024_EPP1342_0001_0017.A_0031_EPP1816_0003_0016.DIG_Inputs_Channel_2.TxPDO_Toggle <-> DIG Inputs Channel 2/TxPDO Toggle
//     PlcTask Inputs/GVL_iXlinker.EtherCAT_Master_EPPxxxx.Beckhoff_EPP1xxx.Beckhoff_EPP1xxxEK1122.A_0018_EPP1321_0060_0016.A_0019_EPP1322_0001_0016.A_0020_EPP1322_0001_0017.A_0021_EPP1332_0001_0016.A_0022_EPP1332_0001_0017.A_0023_EPP1342_0001_0016.A_0024_EPP1342_0001_0017.A_0031_EPP1816_0003_0016.WcState.WcState <-> WcState/WcState
//     PlcTask Inputs/GVL_iXlinker.EtherCAT_Master_EPPxxxx.Beckhoff_EPP1xxx.Beckhoff_EPP1xxxEK1122.A_0018_EPP1321_0060_0016.A_0019_EPP1322_0001_0016.A_0020_EPP1322_0001_0017.A_0021_EPP1332_0001_0016.A_0022_EPP1332_0001_0017.A_0023_EPP1342_0001_0016.A_0024_EPP1342_0001_0017.A_0031_EPP1816_0003_0016.WcState.InputToggle <-> WcState/InputToggle
//     PlcTask Inputs/GVL_iXlinker.EtherCAT_Master_EPPxxxx.Beckhoff_EPP1xxx.Beckhoff_EPP1xxxEK1122.A_0018_EPP1321_0060_0016.A_0019_EPP1322_0001_0016.A_0020_EPP1322_0001_0017.A_0021_EPP1332_0001_0016.A_0022_EPP1332_0001_0017.A_0023_EPP1342_0001_0016.A_0024_EPP1342_0001_0017.A_0031_EPP1816_0003_0016.InfoData.AdsAddr <-> InfoData/AdsAddr
//     PlcTask Inputs/GVL_iXlinker.EtherCAT_Master_EPPxxxx.Beckhoff_EPP1xxx.Beckhoff_EPP1xxxEK1122.A_0018_EPP1321_0060_0016.A_0019_EPP1322_0001_0016.A_0020_EPP1322_0001_0017.A_0021_EPP1332_0001_0016.A_0022_EPP1332_0001_0017.A_0023_EPP1342_0001_0016.A_0024_EPP1342_0001_0017.A_0031_EPP1816_0003_0016.InfoData.State <-> InfoData/State
//   PLC/PLC Instance <-> EtherCAT Master EPPxxxx/Beckhoff EPP1xxx/Beckhoff EPP1xxxEK1122/A_0018(EPP1321-0060-0016)/A_0019(EPP1322-0001-0016)/A_0020(EPP1322-0001-0017)/A_0021(EPP1332-0001-0016)/A_0022(EPP1332-0001-0017)/A_0023(EPP1342-0001-0016)/A_0024(EPP1342-0001-0017)/A_0032(EPP1816-0008-0016)
//     PlcTask Inputs/GVL_iXlinker.EtherCAT_Master_EPPxxxx.Beckhoff_EPP1xxx.Beckhoff_EPP1xxxEK1122.A_0018_EPP1321_0060_0016.A_0019_EPP1322_0001_0016.A_0020_EPP1322_0001_0017.A_0021_EPP1332_0001_0016.A_0022_EPP1332_0001_0017.A_0023_EPP1342_0001_0016.A_0024_EPP1342_0001_0017.A_0032_EPP1816_0008_0016.DIG_Inputs_Channel_1.Input[0] <-> DIG Inputs Channel 1/Input 1
//     PlcTask Inputs/GVL_iXlinker.EtherCAT_Master_EPPxxxx.Beckhoff_EPP1xxx.Beckhoff_EPP1xxxEK1122.A_0018_EPP1321_0060_0016.A_0019_EPP1322_0001_0016.A_0020_EPP1322_0001_0017.A_0021_EPP1332_0001_0016.A_0022_EPP1332_0001_0017.A_0023_EPP1342_0001_0016.A_0024_EPP1342_0001_0017.A_0032_EPP1816_0008_0016.DIG_Inputs_Channel_1.Input[1] <-> DIG Inputs Channel 1/Input 2
//     PlcTask Inputs/GVL_iXlinker.EtherCAT_Master_EPPxxxx.Beckhoff_EPP1xxx.Beckhoff_EPP1xxxEK1122.A_0018_EPP1321_0060_0016.A_0019_EPP1322_0001_0016.A_0020_EPP1322_0001_0017.A_0021_EPP1332_0001_0016.A_0022_EPP1332_0001_0017.A_0023_EPP1342_0001_0016.A_0024_EPP1342_0001_0017.A_0032_EPP1816_0008_0016.DIG_Inputs_Channel_1.Input[2] <-> DIG Inputs Channel 1/Input 3
//     PlcTask Inputs/GVL_iXlinker.EtherCAT_Master_EPPxxxx.Beckhoff_EPP1xxx.Beckhoff_EPP1xxxEK1122.A_0018_EPP1321_0060_0016.A_0019_EPP1322_0001_0016.A_0020_EPP1322_0001_0017.A_0021_EPP1332_0001_0016.A_0022_EPP1332_0001_0017.A_0023_EPP1342_0001_0016.A_0024_EPP1342_0001_0017.A_0032_EPP1816_0008_0016.DIG_Inputs_Channel_1.Input[3] <-> DIG Inputs Channel 1/Input 4
//     PlcTask Inputs/GVL_iXlinker.EtherCAT_Master_EPPxxxx.Beckhoff_EPP1xxx.Beckhoff_EPP1xxxEK1122.A_0018_EPP1321_0060_0016.A_0019_EPP1322_0001_0016.A_0020_EPP1322_0001_0017.A_0021_EPP1332_0001_0016.A_0022_EPP1332_0001_0017.A_0023_EPP1342_0001_0016.A_0024_EPP1342_0001_0017.A_0032_EPP1816_0008_0016.DIG_Inputs_Channel_1.Input[4] <-> DIG Inputs Channel 1/Input 5
//     PlcTask Inputs/GVL_iXlinker.EtherCAT_Master_EPPxxxx.Beckhoff_EPP1xxx.Beckhoff_EPP1xxxEK1122.A_0018_EPP1321_0060_0016.A_0019_EPP1322_0001_0016.A_0020_EPP1322_0001_0017.A_0021_EPP1332_0001_0016.A_0022_EPP1332_0001_0017.A_0023_EPP1342_0001_0016.A_0024_EPP1342_0001_0017.A_0032_EPP1816_0008_0016.DIG_Inputs_Channel_1.Input[5] <-> DIG Inputs Channel 1/Input 6
//     PlcTask Inputs/GVL_iXlinker.EtherCAT_Master_EPPxxxx.Beckhoff_EPP1xxx.Beckhoff_EPP1xxxEK1122.A_0018_EPP1321_0060_0016.A_0019_EPP1322_0001_0016.A_0020_EPP1322_0001_0017.A_0021_EPP1332_0001_0016.A_0022_EPP1332_0001_0017.A_0023_EPP1342_0001_0016.A_0024_EPP1342_0001_0017.A_0032_EPP1816_0008_0016.DIG_Inputs_Channel_1.Input[6] <-> DIG Inputs Channel 1/Input 7
//     PlcTask Inputs/GVL_iXlinker.EtherCAT_Master_EPPxxxx.Beckhoff_EPP1xxx.Beckhoff_EPP1xxxEK1122.A_0018_EPP1321_0060_0016.A_0019_EPP1322_0001_0016.A_0020_EPP1322_0001_0017.A_0021_EPP1332_0001_0016.A_0022_EPP1332_0001_0017.A_0023_EPP1342_0001_0016.A_0024_EPP1342_0001_0017.A_0032_EPP1816_0008_0016.DIG_Inputs_Channel_1.Input[7] <-> DIG Inputs Channel 1/Input 8
//     PlcTask Inputs/GVL_iXlinker.EtherCAT_Master_EPPxxxx.Beckhoff_EPP1xxx.Beckhoff_EPP1xxxEK1122.A_0018_EPP1321_0060_0016.A_0019_EPP1322_0001_0016.A_0020_EPP1322_0001_0017.A_0021_EPP1332_0001_0016.A_0022_EPP1332_0001_0017.A_0023_EPP1342_0001_0016.A_0024_EPP1342_0001_0017.A_0032_EPP1816_0008_0016.DIG_Inputs_Channel_2.Input[0] <-> DIG Inputs Channel 2/Input 1
//     PlcTask Inputs/GVL_iXlinker.EtherCAT_Master_EPPxxxx.Beckhoff_EPP1xxx.Beckhoff_EPP1xxxEK1122.A_0018_EPP1321_0060_0016.A_0019_EPP1322_0001_0016.A_0020_EPP1322_0001_0017.A_0021_EPP1332_0001_0016.A_0022_EPP1332_0001_0017.A_0023_EPP1342_0001_0016.A_0024_EPP1342_0001_0017.A_0032_EPP1816_0008_0016.DIG_Inputs_Channel_2.Input[1] <-> DIG Inputs Channel 2/Input 2
//     PlcTask Inputs/GVL_iXlinker.EtherCAT_Master_EPPxxxx.Beckhoff_EPP1xxx.Beckhoff_EPP1xxxEK1122.A_0018_EPP1321_0060_0016.A_0019_EPP1322_0001_0016.A_0020_EPP1322_0001_0017.A_0021_EPP1332_0001_0016.A_0022_EPP1332_0001_0017.A_0023_EPP1342_0001_0016.A_0024_EPP1342_0001_0017.A_0032_EPP1816_0008_0016.DIG_Inputs_Channel_2.Input[2] <-> DIG Inputs Channel 2/Input 3
//     PlcTask Inputs/GVL_iXlinker.EtherCAT_Master_EPPxxxx.Beckhoff_EPP1xxx.Beckhoff_EPP1xxxEK1122.A_0018_EPP1321_0060_0016.A_0019_EPP1322_0001_0016.A_0020_EPP1322_0001_0017.A_0021_EPP1332_0001_0016.A_0022_EPP1332_0001_0017.A_0023_EPP1342_0001_0016.A_0024_EPP1342_0001_0017.A_0032_EPP1816_0008_0016.DIG_Inputs_Channel_2.Input[3] <-> DIG Inputs Channel 2/Input 4
//     PlcTask Inputs/GVL_iXlinker.EtherCAT_Master_EPPxxxx.Beckhoff_EPP1xxx.Beckhoff_EPP1xxxEK1122.A_0018_EPP1321_0060_0016.A_0019_EPP1322_0001_0016.A_0020_EPP1322_0001_0017.A_0021_EPP1332_0001_0016.A_0022_EPP1332_0001_0017.A_0023_EPP1342_0001_0016.A_0024_EPP1342_0001_0017.A_0032_EPP1816_0008_0016.DIG_Inputs_Channel_2.Input[4] <-> DIG Inputs Channel 2/Input 5
//     PlcTask Inputs/GVL_iXlinker.EtherCAT_Master_EPPxxxx.Beckhoff_EPP1xxx.Beckhoff_EPP1xxxEK1122.A_0018_EPP1321_0060_0016.A_0019_EPP1322_0001_0016.A_0020_EPP1322_0001_0017.A_0021_EPP1332_0001_0016.A_0022_EPP1332_0001_0017.A_0023_EPP1342_0001_0016.A_0024_EPP1342_0001_0017.A_0032_EPP1816_0008_0016.DIG_Inputs_Channel_2.Input[5] <-> DIG Inputs Channel 2/Input 6
//     PlcTask Inputs/GVL_iXlinker.EtherCAT_Master_EPPxxxx.Beckhoff_EPP1xxx.Beckhoff_EPP1xxxEK1122.A_0018_EPP1321_0060_0016.A_0019_EPP1322_0001_0016.A_0020_EPP1322_0001_0017.A_0021_EPP1332_0001_0016.A_0022_EPP1332_0001_0017.A_0023_EPP1342_0001_0016.A_0024_EPP1342_0001_0017.A_0032_EPP1816_0008_0016.DIG_Inputs_Channel_2.Input[6] <-> DIG Inputs Channel 2/Input 7
//     PlcTask Inputs/GVL_iXlinker.EtherCAT_Master_EPPxxxx.Beckhoff_EPP1xxx.Beckhoff_EPP1xxxEK1122.A_0018_EPP1321_0060_0016.A_0019_EPP1322_0001_0016.A_0020_EPP1322_0001_0017.A_0021_EPP1332_0001_0016.A_0022_EPP1332_0001_0017.A_0023_EPP1342_0001_0016.A_0024_EPP1342_0001_0017.A_0032_EPP1816_0008_0016.DIG_Inputs_Channel_2.Input[7] <-> DIG Inputs Channel 2/Input 8
//     PlcTask Inputs/GVL_iXlinker.EtherCAT_Master_EPPxxxx.Beckhoff_EPP1xxx.Beckhoff_EPP1xxxEK1122.A_0018_EPP1321_0060_0016.A_0019_EPP1322_0001_0016.A_0020_EPP1322_0001_0017.A_0021_EPP1332_0001_0016.A_0022_EPP1332_0001_0017.A_0023_EPP1342_0001_0016.A_0024_EPP1342_0001_0017.A_0032_EPP1816_0008_0016.DIG_Inputs_Channel_1.Sync_Error <-> DIG Inputs Channel 1/Sync Error
//     PlcTask Inputs/GVL_iXlinker.EtherCAT_Master_EPPxxxx.Beckhoff_EPP1xxx.Beckhoff_EPP1xxxEK1122.A_0018_EPP1321_0060_0016.A_0019_EPP1322_0001_0016.A_0020_EPP1322_0001_0017.A_0021_EPP1332_0001_0016.A_0022_EPP1332_0001_0017.A_0023_EPP1342_0001_0016.A_0024_EPP1342_0001_0017.A_0032_EPP1816_0008_0016.DIG_Inputs_Channel_2.Sync_Error <-> DIG Inputs Channel 2/Sync Error
//     PlcTask Inputs/GVL_iXlinker.EtherCAT_Master_EPPxxxx.Beckhoff_EPP1xxx.Beckhoff_EPP1xxxEK1122.A_0018_EPP1321_0060_0016.A_0019_EPP1322_0001_0016.A_0020_EPP1322_0001_0017.A_0021_EPP1332_0001_0016.A_0022_EPP1332_0001_0017.A_0023_EPP1342_0001_0016.A_0024_EPP1342_0001_0017.A_0032_EPP1816_0008_0016.WcState.WcState <-> WcState/WcState
//     PlcTask Inputs/GVL_iXlinker.EtherCAT_Master_EPPxxxx.Beckhoff_EPP1xxx.Beckhoff_EPP1xxxEK1122.A_0018_EPP1321_0060_0016.A_0019_EPP1322_0001_0016.A_0020_EPP1322_0001_0017.A_0021_EPP1332_0001_0016.A_0022_EPP1332_0001_0017.A_0023_EPP1342_0001_0016.A_0024_EPP1342_0001_0017.A_0032_EPP1816_0008_0016.WcState.InputToggle <-> WcState/InputToggle
//     PlcTask Inputs/GVL_iXlinker.EtherCAT_Master_EPPxxxx.Beckhoff_EPP1xxx.Beckhoff_EPP1xxxEK1122.A_0018_EPP1321_0060_0016.A_0019_EPP1322_0001_0016.A_0020_EPP1322_0001_0017.A_0021_EPP1332_0001_0016.A_0022_EPP1332_0001_0017.A_0023_EPP1342_0001_0016.A_0024_EPP1342_0001_0017.A_0032_EPP1816_0008_0016.InfoData.AdsAddr <-> InfoData/AdsAddr
//     PlcTask Inputs/GVL_iXlinker.EtherCAT_Master_EPPxxxx.Beckhoff_EPP1xxx.Beckhoff_EPP1xxxEK1122.A_0018_EPP1321_0060_0016.A_0019_EPP1322_0001_0016.A_0020_EPP1322_0001_0017.A_0021_EPP1332_0001_0016.A_0022_EPP1332_0001_0017.A_0023_EPP1342_0001_0016.A_0024_EPP1342_0001_0017.A_0032_EPP1816_0008_0016.InfoData.State <-> InfoData/State
//   PLC/PLC Instance <-> EtherCAT Master EPPxxxx/Beckhoff EPP1xxx/Beckhoff EPP1xxxEK1122/A_0018(EPP1321-0060-0016)/A_0019(EPP1322-0001-0016)/A_0020(EPP1322-0001-0017)/A_0021(EPP1332-0001-0016)/A_0022(EPP1332-0001-0017)/A_0023(EPP1342-0001-0016)/A_0024(EPP1342-0001-0017)/A_0033(EPP1816-0008-0017)
//     PlcTask Inputs/GVL_iXlinker.EtherCAT_Master_EPPxxxx.Beckhoff_EPP1xxx.Beckhoff_EPP1xxxEK1122.A_0018_EPP1321_0060_0016.A_0019_EPP1322_0001_0016.A_0020_EPP1322_0001_0017.A_0021_EPP1332_0001_0016.A_0022_EPP1332_0001_0017.A_0023_EPP1342_0001_0016.A_0024_EPP1342_0001_0017.A_0033_EPP1816_0008_0017.DIG_Inputs_Channel_1.Input[0] <-> DIG Inputs Channel 1/Input 1
//     PlcTask Inputs/GVL_iXlinker.EtherCAT_Master_EPPxxxx.Beckhoff_EPP1xxx.Beckhoff_EPP1xxxEK1122.A_0018_EPP1321_0060_0016.A_0019_EPP1322_0001_0016.A_0020_EPP1322_0001_0017.A_0021_EPP1332_0001_0016.A_0022_EPP1332_0001_0017.A_0023_EPP1342_0001_0016.A_0024_EPP1342_0001_0017.A_0033_EPP1816_0008_0017.DIG_Inputs_Channel_1.Input[1] <-> DIG Inputs Channel 1/Input 2
//     PlcTask Inputs/GVL_iXlinker.EtherCAT_Master_EPPxxxx.Beckhoff_EPP1xxx.Beckhoff_EPP1xxxEK1122.A_0018_EPP1321_0060_0016.A_0019_EPP1322_0001_0016.A_0020_EPP1322_0001_0017.A_0021_EPP1332_0001_0016.A_0022_EPP1332_0001_0017.A_0023_EPP1342_0001_0016.A_0024_EPP1342_0001_0017.A_0033_EPP1816_0008_0017.DIG_Inputs_Channel_1.Input[2] <-> DIG Inputs Channel 1/Input 3
//     PlcTask Inputs/GVL_iXlinker.EtherCAT_Master_EPPxxxx.Beckhoff_EPP1xxx.Beckhoff_EPP1xxxEK1122.A_0018_EPP1321_0060_0016.A_0019_EPP1322_0001_0016.A_0020_EPP1322_0001_0017.A_0021_EPP1332_0001_0016.A_0022_EPP1332_0001_0017.A_0023_EPP1342_0001_0016.A_0024_EPP1342_0001_0017.A_0033_EPP1816_0008_0017.DIG_Inputs_Channel_1.Input[3] <-> DIG Inputs Channel 1/Input 4
//     PlcTask Inputs/GVL_iXlinker.EtherCAT_Master_EPPxxxx.Beckhoff_EPP1xxx.Beckhoff_EPP1xxxEK1122.A_0018_EPP1321_0060_0016.A_0019_EPP1322_0001_0016.A_0020_EPP1322_0001_0017.A_0021_EPP1332_0001_0016.A_0022_EPP1332_0001_0017.A_0023_EPP1342_0001_0016.A_0024_EPP1342_0001_0017.A_0033_EPP1816_0008_0017.DIG_Inputs_Channel_1.Input[4] <-> DIG Inputs Channel 1/Input 5
//     PlcTask Inputs/GVL_iXlinker.EtherCAT_Master_EPPxxxx.Beckhoff_EPP1xxx.Beckhoff_EPP1xxxEK1122.A_0018_EPP1321_0060_0016.A_0019_EPP1322_0001_0016.A_0020_EPP1322_0001_0017.A_0021_EPP1332_0001_0016.A_0022_EPP1332_0001_0017.A_0023_EPP1342_0001_0016.A_0024_EPP1342_0001_0017.A_0033_EPP1816_0008_0017.DIG_Inputs_Channel_1.Input[5] <-> DIG Inputs Channel 1/Input 6
//     PlcTask Inputs/GVL_iXlinker.EtherCAT_Master_EPPxxxx.Beckhoff_EPP1xxx.Beckhoff_EPP1xxxEK1122.A_0018_EPP1321_0060_0016.A_0019_EPP1322_0001_0016.A_0020_EPP1322_0001_0017.A_0021_EPP1332_0001_0016.A_0022_EPP1332_0001_0017.A_0023_EPP1342_0001_0016.A_0024_EPP1342_0001_0017.A_0033_EPP1816_0008_0017.DIG_Inputs_Channel_1.Input[6] <-> DIG Inputs Channel 1/Input 7
//     PlcTask Inputs/GVL_iXlinker.EtherCAT_Master_EPPxxxx.Beckhoff_EPP1xxx.Beckhoff_EPP1xxxEK1122.A_0018_EPP1321_0060_0016.A_0019_EPP1322_0001_0016.A_0020_EPP1322_0001_0017.A_0021_EPP1332_0001_0016.A_0022_EPP1332_0001_0017.A_0023_EPP1342_0001_0016.A_0024_EPP1342_0001_0017.A_0033_EPP1816_0008_0017.DIG_Inputs_Channel_1.Input[7] <-> DIG Inputs Channel 1/Input 8
//     PlcTask Inputs/GVL_iXlinker.EtherCAT_Master_EPPxxxx.Beckhoff_EPP1xxx.Beckhoff_EPP1xxxEK1122.A_0018_EPP1321_0060_0016.A_0019_EPP1322_0001_0016.A_0020_EPP1322_0001_0017.A_0021_EPP1332_0001_0016.A_0022_EPP1332_0001_0017.A_0023_EPP1342_0001_0016.A_0024_EPP1342_0001_0017.A_0033_EPP1816_0008_0017.DIG_Inputs_Channel_2.Input[0] <-> DIG Inputs Channel 2/Input 1
//     PlcTask Inputs/GVL_iXlinker.EtherCAT_Master_EPPxxxx.Beckhoff_EPP1xxx.Beckhoff_EPP1xxxEK1122.A_0018_EPP1321_0060_0016.A_0019_EPP1322_0001_0016.A_0020_EPP1322_0001_0017.A_0021_EPP1332_0001_0016.A_0022_EPP1332_0001_0017.A_0023_EPP1342_0001_0016.A_0024_EPP1342_0001_0017.A_0033_EPP1816_0008_0017.DIG_Inputs_Channel_2.Input[1] <-> DIG Inputs Channel 2/Input 2
//     PlcTask Inputs/GVL_iXlinker.EtherCAT_Master_EPPxxxx.Beckhoff_EPP1xxx.Beckhoff_EPP1xxxEK1122.A_0018_EPP1321_0060_0016.A_0019_EPP1322_0001_0016.A_0020_EPP1322_0001_0017.A_0021_EPP1332_0001_0016.A_0022_EPP1332_0001_0017.A_0023_EPP1342_0001_0016.A_0024_EPP1342_0001_0017.A_0033_EPP1816_0008_0017.DIG_Inputs_Channel_2.Input[2] <-> DIG Inputs Channel 2/Input 3
//     PlcTask Inputs/GVL_iXlinker.EtherCAT_Master_EPPxxxx.Beckhoff_EPP1xxx.Beckhoff_EPP1xxxEK1122.A_0018_EPP1321_0060_0016.A_0019_EPP1322_0001_0016.A_0020_EPP1322_0001_0017.A_0021_EPP1332_0001_0016.A_0022_EPP1332_0001_0017.A_0023_EPP1342_0001_0016.A_0024_EPP1342_0001_0017.A_0033_EPP1816_0008_0017.DIG_Inputs_Channel_2.Input[3] <-> DIG Inputs Channel 2/Input 4
//     PlcTask Inputs/GVL_iXlinker.EtherCAT_Master_EPPxxxx.Beckhoff_EPP1xxx.Beckhoff_EPP1xxxEK1122.A_0018_EPP1321_0060_0016.A_0019_EPP1322_0001_0016.A_0020_EPP1322_0001_0017.A_0021_EPP1332_0001_0016.A_0022_EPP1332_0001_0017.A_0023_EPP1342_0001_0016.A_0024_EPP1342_0001_0017.A_0033_EPP1816_0008_0017.DIG_Inputs_Channel_2.Input[4] <-> DIG Inputs Channel 2/Input 5
//     PlcTask Inputs/GVL_iXlinker.EtherCAT_Master_EPPxxxx.Beckhoff_EPP1xxx.Beckhoff_EPP1xxxEK1122.A_0018_EPP1321_0060_0016.A_0019_EPP1322_0001_0016.A_0020_EPP1322_0001_0017.A_0021_EPP1332_0001_0016.A_0022_EPP1332_0001_0017.A_0023_EPP1342_0001_0016.A_0024_EPP1342_0001_0017.A_0033_EPP1816_0008_0017.DIG_Inputs_Channel_2.Input[5] <-> DIG Inputs Channel 2/Input 6
//     PlcTask Inputs/GVL_iXlinker.EtherCAT_Master_EPPxxxx.Beckhoff_EPP1xxx.Beckhoff_EPP1xxxEK1122.A_0018_EPP1321_0060_0016.A_0019_EPP1322_0001_0016.A_0020_EPP1322_0001_0017.A_0021_EPP1332_0001_0016.A_0022_EPP1332_0001_0017.A_0023_EPP1342_0001_0016.A_0024_EPP1342_0001_0017.A_0033_EPP1816_0008_0017.DIG_Inputs_Channel_2.Input[6] <-> DIG Inputs Channel 2/Input 7
//     PlcTask Inputs/GVL_iXlinker.EtherCAT_Master_EPPxxxx.Beckhoff_EPP1xxx.Beckhoff_EPP1xxxEK1122.A_0018_EPP1321_0060_0016.A_0019_EPP1322_0001_0016.A_0020_EPP1322_0001_0017.A_0021_EPP1332_0001_0016.A_0022_EPP1332_0001_0017.A_0023_EPP1342_0001_0016.A_0024_EPP1342_0001_0017.A_0033_EPP1816_0008_0017.DIG_Inputs_Channel_2.Input[7] <-> DIG Inputs Channel 2/Input 8
//     PlcTask Inputs/GVL_iXlinker.EtherCAT_Master_EPPxxxx.Beckhoff_EPP1xxx.Beckhoff_EPP1xxxEK1122.A_0018_EPP1321_0060_0016.A_0019_EPP1322_0001_0016.A_0020_EPP1322_0001_0017.A_0021_EPP1332_0001_0016.A_0022_EPP1332_0001_0017.A_0023_EPP1342_0001_0016.A_0024_EPP1342_0001_0017.A_0033_EPP1816_0008_0017.DIG_Inputs_Channel_1.Sync_Error <-> DIG Inputs Channel 1/Sync Error
//     PlcTask Inputs/GVL_iXlinker.EtherCAT_Master_EPPxxxx.Beckhoff_EPP1xxx.Beckhoff_EPP1xxxEK1122.A_0018_EPP1321_0060_0016.A_0019_EPP1322_0001_0016.A_0020_EPP1322_0001_0017.A_0021_EPP1332_0001_0016.A_0022_EPP1332_0001_0017.A_0023_EPP1342_0001_0016.A_0024_EPP1342_0001_0017.A_0033_EPP1816_0008_0017.DIG_Inputs_Channel_2.Sync_Error <-> DIG Inputs Channel 2/Sync Error
//     PlcTask Inputs/GVL_iXlinker.EtherCAT_Master_EPPxxxx.Beckhoff_EPP1xxx.Beckhoff_EPP1xxxEK1122.A_0018_EPP1321_0060_0016.A_0019_EPP1322_0001_0016.A_0020_EPP1322_0001_0017.A_0021_EPP1332_0001_0016.A_0022_EPP1332_0001_0017.A_0023_EPP1342_0001_0016.A_0024_EPP1342_0001_0017.A_0033_EPP1816_0008_0017.WcState.WcState <-> WcState/WcState
//     PlcTask Inputs/GVL_iXlinker.EtherCAT_Master_EPPxxxx.Beckhoff_EPP1xxx.Beckhoff_EPP1xxxEK1122.A_0018_EPP1321_0060_0016.A_0019_EPP1322_0001_0016.A_0020_EPP1322_0001_0017.A_0021_EPP1332_0001_0016.A_0022_EPP1332_0001_0017.A_0023_EPP1342_0001_0016.A_0024_EPP1342_0001_0017.A_0033_EPP1816_0008_0017.WcState.InputToggle <-> WcState/InputToggle
//     PlcTask Inputs/GVL_iXlinker.EtherCAT_Master_EPPxxxx.Beckhoff_EPP1xxx.Beckhoff_EPP1xxxEK1122.A_0018_EPP1321_0060_0016.A_0019_EPP1322_0001_0016.A_0020_EPP1322_0001_0017.A_0021_EPP1332_0001_0016.A_0022_EPP1332_0001_0017.A_0023_EPP1342_0001_0016.A_0024_EPP1342_0001_0017.A_0033_EPP1816_0008_0017.InfoData.AdsAddr <-> InfoData/AdsAddr
//     PlcTask Inputs/GVL_iXlinker.EtherCAT_Master_EPPxxxx.Beckhoff_EPP1xxx.Beckhoff_EPP1xxxEK1122.A_0018_EPP1321_0060_0016.A_0019_EPP1322_0001_0016.A_0020_EPP1322_0001_0017.A_0021_EPP1332_0001_0016.A_0022_EPP1332_0001_0017.A_0023_EPP1342_0001_0016.A_0024_EPP1342_0001_0017.A_0033_EPP1816_0008_0017.InfoData.State <-> InfoData/State
//   PLC/PLC Instance <-> EtherCAT Master EPPxxxx/Beckhoff EPP1xxx/Beckhoff EPP1xxxEK1122/A_0018(EPP1321-0060-0016)/A_0019(EPP1322-0001-0016)/A_0020(EPP1322-0001-0017)/A_0021(EPP1332-0001-0016)/A_0022(EPP1332-0001-0017)/A_0023(EPP1342-0001-0016)/A_0024(EPP1342-0001-0017)/A_0034(EPP1816-0008-0018)
//     PlcTask Inputs/GVL_iXlinker.EtherCAT_Master_EPPxxxx.Beckhoff_EPP1xxx.Beckhoff_EPP1xxxEK1122.A_0018_EPP1321_0060_0016.A_0019_EPP1322_0001_0016.A_0020_EPP1322_0001_0017.A_0021_EPP1332_0001_0016.A_0022_EPP1332_0001_0017.A_0023_EPP1342_0001_0016.A_0024_EPP1342_0001_0017.A_0034_EPP1816_0008_0018.DIG_Inputs_Channel_1.Input[0] <-> DIG Inputs Channel 1/Input 1
//     PlcTask Inputs/GVL_iXlinker.EtherCAT_Master_EPPxxxx.Beckhoff_EPP1xxx.Beckhoff_EPP1xxxEK1122.A_0018_EPP1321_0060_0016.A_0019_EPP1322_0001_0016.A_0020_EPP1322_0001_0017.A_0021_EPP1332_0001_0016.A_0022_EPP1332_0001_0017.A_0023_EPP1342_0001_0016.A_0024_EPP1342_0001_0017.A_0034_EPP1816_0008_0018.DIG_Inputs_Channel_1.Input[1] <-> DIG Inputs Channel 1/Input 2
//     PlcTask Inputs/GVL_iXlinker.EtherCAT_Master_EPPxxxx.Beckhoff_EPP1xxx.Beckhoff_EPP1xxxEK1122.A_0018_EPP1321_0060_0016.A_0019_EPP1322_0001_0016.A_0020_EPP1322_0001_0017.A_0021_EPP1332_0001_0016.A_0022_EPP1332_0001_0017.A_0023_EPP1342_0001_0016.A_0024_EPP1342_0001_0017.A_0034_EPP1816_0008_0018.DIG_Inputs_Channel_1.Input[2] <-> DIG Inputs Channel 1/Input 3
//     PlcTask Inputs/GVL_iXlinker.EtherCAT_Master_EPPxxxx.Beckhoff_EPP1xxx.Beckhoff_EPP1xxxEK1122.A_0018_EPP1321_0060_0016.A_0019_EPP1322_0001_0016.A_0020_EPP1322_0001_0017.A_0021_EPP1332_0001_0016.A_0022_EPP1332_0001_0017.A_0023_EPP1342_0001_0016.A_0024_EPP1342_0001_0017.A_0034_EPP1816_0008_0018.DIG_Inputs_Channel_1.Input[3] <-> DIG Inputs Channel 1/Input 4
//     PlcTask Inputs/GVL_iXlinker.EtherCAT_Master_EPPxxxx.Beckhoff_EPP1xxx.Beckhoff_EPP1xxxEK1122.A_0018_EPP1321_0060_0016.A_0019_EPP1322_0001_0016.A_0020_EPP1322_0001_0017.A_0021_EPP1332_0001_0016.A_0022_EPP1332_0001_0017.A_0023_EPP1342_0001_0016.A_0024_EPP1342_0001_0017.A_0034_EPP1816_0008_0018.DIG_Inputs_Channel_1.Input[4] <-> DIG Inputs Channel 1/Input 5
//     PlcTask Inputs/GVL_iXlinker.EtherCAT_Master_EPPxxxx.Beckhoff_EPP1xxx.Beckhoff_EPP1xxxEK1122.A_0018_EPP1321_0060_0016.A_0019_EPP1322_0001_0016.A_0020_EPP1322_0001_0017.A_0021_EPP1332_0001_0016.A_0022_EPP1332_0001_0017.A_0023_EPP1342_0001_0016.A_0024_EPP1342_0001_0017.A_0034_EPP1816_0008_0018.DIG_Inputs_Channel_1.Input[5] <-> DIG Inputs Channel 1/Input 6
//     PlcTask Inputs/GVL_iXlinker.EtherCAT_Master_EPPxxxx.Beckhoff_EPP1xxx.Beckhoff_EPP1xxxEK1122.A_0018_EPP1321_0060_0016.A_0019_EPP1322_0001_0016.A_0020_EPP1322_0001_0017.A_0021_EPP1332_0001_0016.A_0022_EPP1332_0001_0017.A_0023_EPP1342_0001_0016.A_0024_EPP1342_0001_0017.A_0034_EPP1816_0008_0018.DIG_Inputs_Channel_1.Input[6] <-> DIG Inputs Channel 1/Input 7
//     PlcTask Inputs/GVL_iXlinker.EtherCAT_Master_EPPxxxx.Beckhoff_EPP1xxx.Beckhoff_EPP1xxxEK1122.A_0018_EPP1321_0060_0016.A_0019_EPP1322_0001_0016.A_0020_EPP1322_0001_0017.A_0021_EPP1332_0001_0016.A_0022_EPP1332_0001_0017.A_0023_EPP1342_0001_0016.A_0024_EPP1342_0001_0017.A_0034_EPP1816_0008_0018.DIG_Inputs_Channel_1.Input[7] <-> DIG Inputs Channel 1/Input 8
//     PlcTask Inputs/GVL_iXlinker.EtherCAT_Master_EPPxxxx.Beckhoff_EPP1xxx.Beckhoff_EPP1xxxEK1122.A_0018_EPP1321_0060_0016.A_0019_EPP1322_0001_0016.A_0020_EPP1322_0001_0017.A_0021_EPP1332_0001_0016.A_0022_EPP1332_0001_0017.A_0023_EPP1342_0001_0016.A_0024_EPP1342_0001_0017.A_0034_EPP1816_0008_0018.DIG_Inputs_Channel_2.Input[0] <-> DIG Inputs Channel 2/Input 1
//     PlcTask Inputs/GVL_iXlinker.EtherCAT_Master_EPPxxxx.Beckhoff_EPP1xxx.Beckhoff_EPP1xxxEK1122.A_0018_EPP1321_0060_0016.A_0019_EPP1322_0001_0016.A_0020_EPP1322_0001_0017.A_0021_EPP1332_0001_0016.A_0022_EPP1332_0001_0017.A_0023_EPP1342_0001_0016.A_0024_EPP1342_0001_0017.A_0034_EPP1816_0008_0018.DIG_Inputs_Channel_2.Input[1] <-> DIG Inputs Channel 2/Input 2
//     PlcTask Inputs/GVL_iXlinker.EtherCAT_Master_EPPxxxx.Beckhoff_EPP1xxx.Beckhoff_EPP1xxxEK1122.A_0018_EPP1321_0060_0016.A_0019_EPP1322_0001_0016.A_0020_EPP1322_0001_0017.A_0021_EPP1332_0001_0016.A_0022_EPP1332_0001_0017.A_0023_EPP1342_0001_0016.A_0024_EPP1342_0001_0017.A_0034_EPP1816_0008_0018.DIG_Inputs_Channel_2.Input[2] <-> DIG Inputs Channel 2/Input 3
//     PlcTask Inputs/GVL_iXlinker.EtherCAT_Master_EPPxxxx.Beckhoff_EPP1xxx.Beckhoff_EPP1xxxEK1122.A_0018_EPP1321_0060_0016.A_0019_EPP1322_0001_0016.A_0020_EPP1322_0001_0017.A_0021_EPP1332_0001_0016.A_0022_EPP1332_0001_0017.A_0023_EPP1342_0001_0016.A_0024_EPP1342_0001_0017.A_0034_EPP1816_0008_0018.DIG_Inputs_Channel_2.Input[3] <-> DIG Inputs Channel 2/Input 4
//     PlcTask Inputs/GVL_iXlinker.EtherCAT_Master_EPPxxxx.Beckhoff_EPP1xxx.Beckhoff_EPP1xxxEK1122.A_0018_EPP1321_0060_0016.A_0019_EPP1322_0001_0016.A_0020_EPP1322_0001_0017.A_0021_EPP1332_0001_0016.A_0022_EPP1332_0001_0017.A_0023_EPP1342_0001_0016.A_0024_EPP1342_0001_0017.A_0034_EPP1816_0008_0018.DIG_Inputs_Channel_2.Input[4] <-> DIG Inputs Channel 2/Input 5
//     PlcTask Inputs/GVL_iXlinker.EtherCAT_Master_EPPxxxx.Beckhoff_EPP1xxx.Beckhoff_EPP1xxxEK1122.A_0018_EPP1321_0060_0016.A_0019_EPP1322_0001_0016.A_0020_EPP1322_0001_0017.A_0021_EPP1332_0001_0016.A_0022_EPP1332_0001_0017.A_0023_EPP1342_0001_0016.A_0024_EPP1342_0001_0017.A_0034_EPP1816_0008_0018.DIG_Inputs_Channel_2.Input[5] <-> DIG Inputs Channel 2/Input 6
//     PlcTask Inputs/GVL_iXlinker.EtherCAT_Master_EPPxxxx.Beckhoff_EPP1xxx.Beckhoff_EPP1xxxEK1122.A_0018_EPP1321_0060_0016.A_0019_EPP1322_0001_0016.A_0020_EPP1322_0001_0017.A_0021_EPP1332_0001_0016.A_0022_EPP1332_0001_0017.A_0023_EPP1342_0001_0016.A_0024_EPP1342_0001_0017.A_0034_EPP1816_0008_0018.DIG_Inputs_Channel_2.Input[6] <-> DIG Inputs Channel 2/Input 7
//     PlcTask Inputs/GVL_iXlinker.EtherCAT_Master_EPPxxxx.Beckhoff_EPP1xxx.Beckhoff_EPP1xxxEK1122.A_0018_EPP1321_0060_0016.A_0019_EPP1322_0001_0016.A_0020_EPP1322_0001_0017.A_0021_EPP1332_0001_0016.A_0022_EPP1332_0001_0017.A_0023_EPP1342_0001_0016.A_0024_EPP1342_0001_0017.A_0034_EPP1816_0008_0018.DIG_Inputs_Channel_2.Input[7] <-> DIG Inputs Channel 2/Input 8
//     PlcTask Inputs/GVL_iXlinker.EtherCAT_Master_EPPxxxx.Beckhoff_EPP1xxx.Beckhoff_EPP1xxxEK1122.A_0018_EPP1321_0060_0016.A_0019_EPP1322_0001_0016.A_0020_EPP1322_0001_0017.A_0021_EPP1332_0001_0016.A_0022_EPP1332_0001_0017.A_0023_EPP1342_0001_0016.A_0024_EPP1342_0001_0017.A_0034_EPP1816_0008_0018.DIG_Inputs_Channel_1.Sync_error <-> DIG Inputs Channel 1/Sync error
//     PlcTask Inputs/GVL_iXlinker.EtherCAT_Master_EPPxxxx.Beckhoff_EPP1xxx.Beckhoff_EPP1xxxEK1122.A_0018_EPP1321_0060_0016.A_0019_EPP1322_0001_0016.A_0020_EPP1322_0001_0017.A_0021_EPP1332_0001_0016.A_0022_EPP1332_0001_0017.A_0023_EPP1342_0001_0016.A_0024_EPP1342_0001_0017.A_0034_EPP1816_0008_0018.DIG_Inputs_Channel_2.Sync_error <-> DIG Inputs Channel 2/Sync error
//     PlcTask Inputs/GVL_iXlinker.EtherCAT_Master_EPPxxxx.Beckhoff_EPP1xxx.Beckhoff_EPP1xxxEK1122.A_0018_EPP1321_0060_0016.A_0019_EPP1322_0001_0016.A_0020_EPP1322_0001_0017.A_0021_EPP1332_0001_0016.A_0022_EPP1332_0001_0017.A_0023_EPP1342_0001_0016.A_0024_EPP1342_0001_0017.A_0034_EPP1816_0008_0018.DIG_Inputs_Channel_1.TxPDO_Toggle <-> DIG Inputs Channel 1/TxPDO Toggle
//     PlcTask Inputs/GVL_iXlinker.EtherCAT_Master_EPPxxxx.Beckhoff_EPP1xxx.Beckhoff_EPP1xxxEK1122.A_0018_EPP1321_0060_0016.A_0019_EPP1322_0001_0016.A_0020_EPP1322_0001_0017.A_0021_EPP1332_0001_0016.A_0022_EPP1332_0001_0017.A_0023_EPP1342_0001_0016.A_0024_EPP1342_0001_0017.A_0034_EPP1816_0008_0018.DIG_Inputs_Channel_2.TxPDO_Toggle <-> DIG Inputs Channel 2/TxPDO Toggle
//     PlcTask Inputs/GVL_iXlinker.EtherCAT_Master_EPPxxxx.Beckhoff_EPP1xxx.Beckhoff_EPP1xxxEK1122.A_0018_EPP1321_0060_0016.A_0019_EPP1322_0001_0016.A_0020_EPP1322_0001_0017.A_0021_EPP1332_0001_0016.A_0022_EPP1332_0001_0017.A_0023_EPP1342_0001_0016.A_0024_EPP1342_0001_0017.A_0034_EPP1816_0008_0018.WcState.WcState <-> WcState/WcState
//     PlcTask Inputs/GVL_iXlinker.EtherCAT_Master_EPPxxxx.Beckhoff_EPP1xxx.Beckhoff_EPP1xxxEK1122.A_0018_EPP1321_0060_0016.A_0019_EPP1322_0001_0016.A_0020_EPP1322_0001_0017.A_0021_EPP1332_0001_0016.A_0022_EPP1332_0001_0017.A_0023_EPP1342_0001_0016.A_0024_EPP1342_0001_0017.A_0034_EPP1816_0008_0018.WcState.InputToggle <-> WcState/InputToggle
//     PlcTask Inputs/GVL_iXlinker.EtherCAT_Master_EPPxxxx.Beckhoff_EPP1xxx.Beckhoff_EPP1xxxEK1122.A_0018_EPP1321_0060_0016.A_0019_EPP1322_0001_0016.A_0020_EPP1322_0001_0017.A_0021_EPP1332_0001_0016.A_0022_EPP1332_0001_0017.A_0023_EPP1342_0001_0016.A_0024_EPP1342_0001_0017.A_0034_EPP1816_0008_0018.InfoData.AdsAddr <-> InfoData/AdsAddr
//     PlcTask Inputs/GVL_iXlinker.EtherCAT_Master_EPPxxxx.Beckhoff_EPP1xxx.Beckhoff_EPP1xxxEK1122.A_0018_EPP1321_0060_0016.A_0019_EPP1322_0001_0016.A_0020_EPP1322_0001_0017.A_0021_EPP1332_0001_0016.A_0022_EPP1332_0001_0017.A_0023_EPP1342_0001_0016.A_0024_EPP1342_0001_0017.A_0034_EPP1816_0008_0018.InfoData.State <-> InfoData/State
//   PLC/PLC Instance <-> EtherCAT Master EPPxxxx/Beckhoff EPP1xxx/Beckhoff EPP1xxxEK1122/A_0018(EPP1321-0060-0016)/A_0019(EPP1322-0001-0016)/A_0020(EPP1322-0001-0017)/A_0021(EPP1332-0001-0016)/A_0022(EPP1332-0001-0017)/A_0023(EPP1342-0001-0016)/A_0024(EPP1342-0001-0017)/A_0035(EPP1816-3008-0016)
//     PlcTask Inputs/GVL_iXlinker.EtherCAT_Master_EPPxxxx.Beckhoff_EPP1xxx.Beckhoff_EPP1xxxEK1122.A_0018_EPP1321_0060_0016.A_0019_EPP1322_0001_0016.A_0020_EPP1322_0001_0017.A_0021_EPP1332_0001_0016.A_0022_EPP1332_0001_0017.A_0023_EPP1342_0001_0016.A_0024_EPP1342_0001_0017.A_0035_EPP1816_3008_0016.DIG_Inputs_Channel_1.Input[0] <-> DIG Inputs Channel 1/Input 1
//     PlcTask Inputs/GVL_iXlinker.EtherCAT_Master_EPPxxxx.Beckhoff_EPP1xxx.Beckhoff_EPP1xxxEK1122.A_0018_EPP1321_0060_0016.A_0019_EPP1322_0001_0016.A_0020_EPP1322_0001_0017.A_0021_EPP1332_0001_0016.A_0022_EPP1332_0001_0017.A_0023_EPP1342_0001_0016.A_0024_EPP1342_0001_0017.A_0035_EPP1816_3008_0016.DIG_Inputs_Channel_1.Input[1] <-> DIG Inputs Channel 1/Input 2
//     PlcTask Inputs/GVL_iXlinker.EtherCAT_Master_EPPxxxx.Beckhoff_EPP1xxx.Beckhoff_EPP1xxxEK1122.A_0018_EPP1321_0060_0016.A_0019_EPP1322_0001_0016.A_0020_EPP1322_0001_0017.A_0021_EPP1332_0001_0016.A_0022_EPP1332_0001_0017.A_0023_EPP1342_0001_0016.A_0024_EPP1342_0001_0017.A_0035_EPP1816_3008_0016.DIG_Inputs_Channel_1.Input[2] <-> DIG Inputs Channel 1/Input 3
//     PlcTask Inputs/GVL_iXlinker.EtherCAT_Master_EPPxxxx.Beckhoff_EPP1xxx.Beckhoff_EPP1xxxEK1122.A_0018_EPP1321_0060_0016.A_0019_EPP1322_0001_0016.A_0020_EPP1322_0001_0017.A_0021_EPP1332_0001_0016.A_0022_EPP1332_0001_0017.A_0023_EPP1342_0001_0016.A_0024_EPP1342_0001_0017.A_0035_EPP1816_3008_0016.DIG_Inputs_Channel_1.Input[3] <-> DIG Inputs Channel 1/Input 4
//     PlcTask Inputs/GVL_iXlinker.EtherCAT_Master_EPPxxxx.Beckhoff_EPP1xxx.Beckhoff_EPP1xxxEK1122.A_0018_EPP1321_0060_0016.A_0019_EPP1322_0001_0016.A_0020_EPP1322_0001_0017.A_0021_EPP1332_0001_0016.A_0022_EPP1332_0001_0017.A_0023_EPP1342_0001_0016.A_0024_EPP1342_0001_0017.A_0035_EPP1816_3008_0016.DIG_Inputs_Channel_1.Input[4] <-> DIG Inputs Channel 1/Input 5
//     PlcTask Inputs/GVL_iXlinker.EtherCAT_Master_EPPxxxx.Beckhoff_EPP1xxx.Beckhoff_EPP1xxxEK1122.A_0018_EPP1321_0060_0016.A_0019_EPP1322_0001_0016.A_0020_EPP1322_0001_0017.A_0021_EPP1332_0001_0016.A_0022_EPP1332_0001_0017.A_0023_EPP1342_0001_0016.A_0024_EPP1342_0001_0017.A_0035_EPP1816_3008_0016.DIG_Inputs_Channel_1.Input[5] <-> DIG Inputs Channel 1/Input 6
//     PlcTask Inputs/GVL_iXlinker.EtherCAT_Master_EPPxxxx.Beckhoff_EPP1xxx.Beckhoff_EPP1xxxEK1122.A_0018_EPP1321_0060_0016.A_0019_EPP1322_0001_0016.A_0020_EPP1322_0001_0017.A_0021_EPP1332_0001_0016.A_0022_EPP1332_0001_0017.A_0023_EPP1342_0001_0016.A_0024_EPP1342_0001_0017.A_0035_EPP1816_3008_0016.DIG_Inputs_Channel_1.Input[6] <-> DIG Inputs Channel 1/Input 7
//     PlcTask Inputs/GVL_iXlinker.EtherCAT_Master_EPPxxxx.Beckhoff_EPP1xxx.Beckhoff_EPP1xxxEK1122.A_0018_EPP1321_0060_0016.A_0019_EPP1322_0001_0016.A_0020_EPP1322_0001_0017.A_0021_EPP1332_0001_0016.A_0022_EPP1332_0001_0017.A_0023_EPP1342_0001_0016.A_0024_EPP1342_0001_0017.A_0035_EPP1816_3008_0016.DIG_Inputs_Channel_1.Input[7] <-> DIG Inputs Channel 1/Input 8
//     PlcTask Inputs/GVL_iXlinker.EtherCAT_Master_EPPxxxx.Beckhoff_EPP1xxx.Beckhoff_EPP1xxxEK1122.A_0018_EPP1321_0060_0016.A_0019_EPP1322_0001_0016.A_0020_EPP1322_0001_0017.A_0021_EPP1332_0001_0016.A_0022_EPP1332_0001_0017.A_0023_EPP1342_0001_0016.A_0024_EPP1342_0001_0017.A_0035_EPP1816_3008_0016.DIG_Inputs_Channel_2.Input[0] <-> DIG Inputs Channel 2/Input 1
//     PlcTask Inputs/GVL_iXlinker.EtherCAT_Master_EPPxxxx.Beckhoff_EPP1xxx.Beckhoff_EPP1xxxEK1122.A_0018_EPP1321_0060_0016.A_0019_EPP1322_0001_0016.A_0020_EPP1322_0001_0017.A_0021_EPP1332_0001_0016.A_0022_EPP1332_0001_0017.A_0023_EPP1342_0001_0016.A_0024_EPP1342_0001_0017.A_0035_EPP1816_3008_0016.DIG_Inputs_Channel_2.Input[1] <-> DIG Inputs Channel 2/Input 2
//     PlcTask Inputs/GVL_iXlinker.EtherCAT_Master_EPPxxxx.Beckhoff_EPP1xxx.Beckhoff_EPP1xxxEK1122.A_0018_EPP1321_0060_0016.A_0019_EPP1322_0001_0016.A_0020_EPP1322_0001_0017.A_0021_EPP1332_0001_0016.A_0022_EPP1332_0001_0017.A_0023_EPP1342_0001_0016.A_0024_EPP1342_0001_0017.A_0035_EPP1816_3008_0016.DIG_Inputs_Channel_2.Input[2] <-> DIG Inputs Channel 2/Input 3
//     PlcTask Inputs/GVL_iXlinker.EtherCAT_Master_EPPxxxx.Beckhoff_EPP1xxx.Beckhoff_EPP1xxxEK1122.A_0018_EPP1321_0060_0016.A_0019_EPP1322_0001_0016.A_0020_EPP1322_0001_0017.A_0021_EPP1332_0001_0016.A_0022_EPP1332_0001_0017.A_0023_EPP1342_0001_0016.A_0024_EPP1342_0001_0017.A_0035_EPP1816_3008_0016.DIG_Inputs_Channel_2.Input[3] <-> DIG Inputs Channel 2/Input 4
//     PlcTask Inputs/GVL_iXlinker.EtherCAT_Master_EPPxxxx.Beckhoff_EPP1xxx.Beckhoff_EPP1xxxEK1122.A_0018_EPP1321_0060_0016.A_0019_EPP1322_0001_0016.A_0020_EPP1322_0001_0017.A_0021_EPP1332_0001_0016.A_0022_EPP1332_0001_0017.A_0023_EPP1342_0001_0016.A_0024_EPP1342_0001_0017.A_0035_EPP1816_3008_0016.DIG_Inputs_Channel_2.Input[4] <-> DIG Inputs Channel 2/Input 5
//     PlcTask Inputs/GVL_iXlinker.EtherCAT_Master_EPPxxxx.Beckhoff_EPP1xxx.Beckhoff_EPP1xxxEK1122.A_0018_EPP1321_0060_0016.A_0019_EPP1322_0001_0016.A_0020_EPP1322_0001_0017.A_0021_EPP1332_0001_0016.A_0022_EPP1332_0001_0017.A_0023_EPP1342_0001_0016.A_0024_EPP1342_0001_0017.A_0035_EPP1816_3008_0016.DIG_Inputs_Channel_2.Input[5] <-> DIG Inputs Channel 2/Input 6
//     PlcTask Inputs/GVL_iXlinker.EtherCAT_Master_EPPxxxx.Beckhoff_EPP1xxx.Beckhoff_EPP1xxxEK1122.A_0018_EPP1321_0060_0016.A_0019_EPP1322_0001_0016.A_0020_EPP1322_0001_0017.A_0021_EPP1332_0001_0016.A_0022_EPP1332_0001_0017.A_0023_EPP1342_0001_0016.A_0024_EPP1342_0001_0017.A_0035_EPP1816_3008_0016.DIG_Inputs_Channel_2.Input[6] <-> DIG Inputs Channel 2/Input 7
//     PlcTask Inputs/GVL_iXlinker.EtherCAT_Master_EPPxxxx.Beckhoff_EPP1xxx.Beckhoff_EPP1xxxEK1122.A_0018_EPP1321_0060_0016.A_0019_EPP1322_0001_0016.A_0020_EPP1322_0001_0017.A_0021_EPP1332_0001_0016.A_0022_EPP1332_0001_0017.A_0023_EPP1342_0001_0016.A_0024_EPP1342_0001_0017.A_0035_EPP1816_3008_0016.DIG_Inputs_Channel_2.Input[7] <-> DIG Inputs Channel 2/Input 8
//     PlcTask Inputs/GVL_iXlinker.EtherCAT_Master_EPPxxxx.Beckhoff_EPP1xxx.Beckhoff_EPP1xxxEK1122.A_0018_EPP1321_0060_0016.A_0019_EPP1322_0001_0016.A_0020_EPP1322_0001_0017.A_0021_EPP1332_0001_0016.A_0022_EPP1332_0001_0017.A_0023_EPP1342_0001_0016.A_0024_EPP1342_0001_0017.A_0035_EPP1816_3008_0016.AI_Inputs_Channel_1.Status/Error <-> AI Inputs Channel 1/Status/Error
//     PlcTask Inputs/GVL_iXlinker.EtherCAT_Master_EPPxxxx.Beckhoff_EPP1xxx.Beckhoff_EPP1xxxEK1122.A_0018_EPP1321_0060_0016.A_0019_EPP1322_0001_0016.A_0020_EPP1322_0001_0017.A_0021_EPP1332_0001_0016.A_0022_EPP1332_0001_0017.A_0023_EPP1342_0001_0016.A_0024_EPP1342_0001_0017.A_0035_EPP1816_3008_0016.AI_Inputs_Channel_2.Status/Error <-> AI Inputs Channel 2/Status/Error
//     PlcTask Inputs/GVL_iXlinker.EtherCAT_Master_EPPxxxx.Beckhoff_EPP1xxx.Beckhoff_EPP1xxxEK1122.A_0018_EPP1321_0060_0016.A_0019_EPP1322_0001_0016.A_0020_EPP1322_0001_0017.A_0021_EPP1332_0001_0016.A_0022_EPP1332_0001_0017.A_0023_EPP1342_0001_0016.A_0024_EPP1342_0001_0017.A_0035_EPP1816_3008_0016.AI_Inputs_Channel_3.Status/Error <-> AI Inputs Channel 3/Status/Error
//     PlcTask Inputs/GVL_iXlinker.EtherCAT_Master_EPPxxxx.Beckhoff_EPP1xxx.Beckhoff_EPP1xxxEK1122.A_0018_EPP1321_0060_0016.A_0019_EPP1322_0001_0016.A_0020_EPP1322_0001_0017.A_0021_EPP1332_0001_0016.A_0022_EPP1332_0001_0017.A_0023_EPP1342_0001_0016.A_0024_EPP1342_0001_0017.A_0035_EPP1816_3008_0016.AI_Inputs_Channel_4.Status/Error <-> AI Inputs Channel 4/Status/Error
//     PlcTask Inputs/GVL_iXlinker.EtherCAT_Master_EPPxxxx.Beckhoff_EPP1xxx.Beckhoff_EPP1xxxEK1122.A_0018_EPP1321_0060_0016.A_0019_EPP1322_0001_0016.A_0020_EPP1322_0001_0017.A_0021_EPP1332_0001_0016.A_0022_EPP1332_0001_0017.A_0023_EPP1342_0001_0016.A_0024_EPP1342_0001_0017.A_0035_EPP1816_3008_0016.AI_Inputs_Channel_5.Status/Error <-> AI Inputs Channel 5/Status/Error
//     PlcTask Inputs/GVL_iXlinker.EtherCAT_Master_EPPxxxx.Beckhoff_EPP1xxx.Beckhoff_EPP1xxxEK1122.A_0018_EPP1321_0060_0016.A_0019_EPP1322_0001_0016.A_0020_EPP1322_0001_0017.A_0021_EPP1332_0001_0016.A_0022_EPP1332_0001_0017.A_0023_EPP1342_0001_0016.A_0024_EPP1342_0001_0017.A_0035_EPP1816_3008_0016.AI_Inputs_Channel_6.Status/Error <-> AI Inputs Channel 6/Status/Error
//     PlcTask Inputs/GVL_iXlinker.EtherCAT_Master_EPPxxxx.Beckhoff_EPP1xxx.Beckhoff_EPP1xxxEK1122.A_0018_EPP1321_0060_0016.A_0019_EPP1322_0001_0016.A_0020_EPP1322_0001_0017.A_0021_EPP1332_0001_0016.A_0022_EPP1332_0001_0017.A_0023_EPP1342_0001_0016.A_0024_EPP1342_0001_0017.A_0035_EPP1816_3008_0016.AI_Inputs_Channel_1.Status/TxPDO_Toggle <-> AI Inputs Channel 1/Status/TxPDO Toggle
//     PlcTask Inputs/GVL_iXlinker.EtherCAT_Master_EPPxxxx.Beckhoff_EPP1xxx.Beckhoff_EPP1xxxEK1122.A_0018_EPP1321_0060_0016.A_0019_EPP1322_0001_0016.A_0020_EPP1322_0001_0017.A_0021_EPP1332_0001_0016.A_0022_EPP1332_0001_0017.A_0023_EPP1342_0001_0016.A_0024_EPP1342_0001_0017.A_0035_EPP1816_3008_0016.AI_Inputs_Channel_2.Status/TxPDO_Toggle <-> AI Inputs Channel 2/Status/TxPDO Toggle
//     PlcTask Inputs/GVL_iXlinker.EtherCAT_Master_EPPxxxx.Beckhoff_EPP1xxx.Beckhoff_EPP1xxxEK1122.A_0018_EPP1321_0060_0016.A_0019_EPP1322_0001_0016.A_0020_EPP1322_0001_0017.A_0021_EPP1332_0001_0016.A_0022_EPP1332_0001_0017.A_0023_EPP1342_0001_0016.A_0024_EPP1342_0001_0017.A_0035_EPP1816_3008_0016.AI_Inputs_Channel_3.Status/TxPDO_Toggle <-> AI Inputs Channel 3/Status/TxPDO Toggle
//     PlcTask Inputs/GVL_iXlinker.EtherCAT_Master_EPPxxxx.Beckhoff_EPP1xxx.Beckhoff_EPP1xxxEK1122.A_0018_EPP1321_0060_0016.A_0019_EPP1322_0001_0016.A_0020_EPP1322_0001_0017.A_0021_EPP1332_0001_0016.A_0022_EPP1332_0001_0017.A_0023_EPP1342_0001_0016.A_0024_EPP1342_0001_0017.A_0035_EPP1816_3008_0016.AI_Inputs_Channel_4.Status/TxPDO_Toggle <-> AI Inputs Channel 4/Status/TxPDO Toggle
//     PlcTask Inputs/GVL_iXlinker.EtherCAT_Master_EPPxxxx.Beckhoff_EPP1xxx.Beckhoff_EPP1xxxEK1122.A_0018_EPP1321_0060_0016.A_0019_EPP1322_0001_0016.A_0020_EPP1322_0001_0017.A_0021_EPP1332_0001_0016.A_0022_EPP1332_0001_0017.A_0023_EPP1342_0001_0016.A_0024_EPP1342_0001_0017.A_0035_EPP1816_3008_0016.AI_Inputs_Channel_5.Status/TxPDO_Toggle <-> AI Inputs Channel 5/Status/TxPDO Toggle
//     PlcTask Inputs/GVL_iXlinker.EtherCAT_Master_EPPxxxx.Beckhoff_EPP1xxx.Beckhoff_EPP1xxxEK1122.A_0018_EPP1321_0060_0016.A_0019_EPP1322_0001_0016.A_0020_EPP1322_0001_0017.A_0021_EPP1332_0001_0016.A_0022_EPP1332_0001_0017.A_0023_EPP1342_0001_0016.A_0024_EPP1342_0001_0017.A_0035_EPP1816_3008_0016.AI_Inputs_Channel_6.Status/TxPDO_Toggle <-> AI Inputs Channel 6/Status/TxPDO Toggle
//     PlcTask Inputs/GVL_iXlinker.EtherCAT_Master_EPPxxxx.Beckhoff_EPP1xxx.Beckhoff_EPP1xxxEK1122.A_0018_EPP1321_0060_0016.A_0019_EPP1322_0001_0016.A_0020_EPP1322_0001_0017.A_0021_EPP1332_0001_0016.A_0022_EPP1332_0001_0017.A_0023_EPP1342_0001_0016.A_0024_EPP1342_0001_0017.A_0035_EPP1816_3008_0016.AI_Inputs_Channel_1.Value <-> AI Inputs Channel 1/Value
//     PlcTask Inputs/GVL_iXlinker.EtherCAT_Master_EPPxxxx.Beckhoff_EPP1xxx.Beckhoff_EPP1xxxEK1122.A_0018_EPP1321_0060_0016.A_0019_EPP1322_0001_0016.A_0020_EPP1322_0001_0017.A_0021_EPP1332_0001_0016.A_0022_EPP1332_0001_0017.A_0023_EPP1342_0001_0016.A_0024_EPP1342_0001_0017.A_0035_EPP1816_3008_0016.AI_Inputs_Channel_2.Value <-> AI Inputs Channel 2/Value
//     PlcTask Inputs/GVL_iXlinker.EtherCAT_Master_EPPxxxx.Beckhoff_EPP1xxx.Beckhoff_EPP1xxxEK1122.A_0018_EPP1321_0060_0016.A_0019_EPP1322_0001_0016.A_0020_EPP1322_0001_0017.A_0021_EPP1332_0001_0016.A_0022_EPP1332_0001_0017.A_0023_EPP1342_0001_0016.A_0024_EPP1342_0001_0017.A_0035_EPP1816_3008_0016.AI_Inputs_Channel_3.Value <-> AI Inputs Channel 3/Value
//     PlcTask Inputs/GVL_iXlinker.EtherCAT_Master_EPPxxxx.Beckhoff_EPP1xxx.Beckhoff_EPP1xxxEK1122.A_0018_EPP1321_0060_0016.A_0019_EPP1322_0001_0016.A_0020_EPP1322_0001_0017.A_0021_EPP1332_0001_0016.A_0022_EPP1332_0001_0017.A_0023_EPP1342_0001_0016.A_0024_EPP1342_0001_0017.A_0035_EPP1816_3008_0016.AI_Inputs_Channel_4.Value <-> AI Inputs Channel 4/Value
//     PlcTask Inputs/GVL_iXlinker.EtherCAT_Master_EPPxxxx.Beckhoff_EPP1xxx.Beckhoff_EPP1xxxEK1122.A_0018_EPP1321_0060_0016.A_0019_EPP1322_0001_0016.A_0020_EPP1322_0001_0017.A_0021_EPP1332_0001_0016.A_0022_EPP1332_0001_0017.A_0023_EPP1342_0001_0016.A_0024_EPP1342_0001_0017.A_0035_EPP1816_3008_0016.AI_Inputs_Channel_5.Value <-> AI Inputs Channel 5/Value
//     PlcTask Inputs/GVL_iXlinker.EtherCAT_Master_EPPxxxx.Beckhoff_EPP1xxx.Beckhoff_EPP1xxxEK1122.A_0018_EPP1321_0060_0016.A_0019_EPP1322_0001_0016.A_0020_EPP1322_0001_0017.A_0021_EPP1332_0001_0016.A_0022_EPP1332_0001_0017.A_0023_EPP1342_0001_0016.A_0024_EPP1342_0001_0017.A_0035_EPP1816_3008_0016.AI_Inputs_Channel_6.Value <-> AI Inputs Channel 6/Value
//     PlcTask Inputs/GVL_iXlinker.EtherCAT_Master_EPPxxxx.Beckhoff_EPP1xxx.Beckhoff_EPP1xxxEK1122.A_0018_EPP1321_0060_0016.A_0019_EPP1322_0001_0016.A_0020_EPP1322_0001_0017.A_0021_EPP1332_0001_0016.A_0022_EPP1332_0001_0017.A_0023_EPP1342_0001_0016.A_0024_EPP1342_0001_0017.A_0035_EPP1816_3008_0016.DIG_Inputs_Device.Us_Undervoltage <-> DIG Inputs Device/Us Undervoltage
//     PlcTask Inputs/GVL_iXlinker.EtherCAT_Master_EPPxxxx.Beckhoff_EPP1xxx.Beckhoff_EPP1xxxEK1122.A_0018_EPP1321_0060_0016.A_0019_EPP1322_0001_0016.A_0020_EPP1322_0001_0017.A_0021_EPP1332_0001_0016.A_0022_EPP1332_0001_0017.A_0023_EPP1342_0001_0016.A_0024_EPP1342_0001_0017.A_0035_EPP1816_3008_0016.DIG_Inputs_Device.Up_Undervoltage <-> DIG Inputs Device/Up Undervoltage
//     PlcTask Inputs/GVL_iXlinker.EtherCAT_Master_EPPxxxx.Beckhoff_EPP1xxx.Beckhoff_EPP1xxxEK1122.A_0018_EPP1321_0060_0016.A_0019_EPP1322_0001_0016.A_0020_EPP1322_0001_0017.A_0021_EPP1332_0001_0016.A_0022_EPP1332_0001_0017.A_0023_EPP1342_0001_0016.A_0024_EPP1342_0001_0017.A_0035_EPP1816_3008_0016.DIG_Inputs_Device.Sync_error <-> DIG Inputs Device/Sync error
//     PlcTask Inputs/GVL_iXlinker.EtherCAT_Master_EPPxxxx.Beckhoff_EPP1xxx.Beckhoff_EPP1xxxEK1122.A_0018_EPP1321_0060_0016.A_0019_EPP1322_0001_0016.A_0020_EPP1322_0001_0017.A_0021_EPP1332_0001_0016.A_0022_EPP1332_0001_0017.A_0023_EPP1342_0001_0016.A_0024_EPP1342_0001_0017.A_0035_EPP1816_3008_0016.DIG_Inputs_Device.TxPDO_Toggle <-> DIG Inputs Device/TxPDO Toggle
//     PlcTask Inputs/GVL_iXlinker.EtherCAT_Master_EPPxxxx.Beckhoff_EPP1xxx.Beckhoff_EPP1xxxEK1122.A_0018_EPP1321_0060_0016.A_0019_EPP1322_0001_0016.A_0020_EPP1322_0001_0017.A_0021_EPP1332_0001_0016.A_0022_EPP1332_0001_0017.A_0023_EPP1342_0001_0016.A_0024_EPP1342_0001_0017.A_0035_EPP1816_3008_0016.WcState.WcState <-> WcState/WcState
//     PlcTask Inputs/GVL_iXlinker.EtherCAT_Master_EPPxxxx.Beckhoff_EPP1xxx.Beckhoff_EPP1xxxEK1122.A_0018_EPP1321_0060_0016.A_0019_EPP1322_0001_0016.A_0020_EPP1322_0001_0017.A_0021_EPP1332_0001_0016.A_0022_EPP1332_0001_0017.A_0023_EPP1342_0001_0016.A_0024_EPP1342_0001_0017.A_0035_EPP1816_3008_0016.WcState.InputToggle <-> WcState/InputToggle
//     PlcTask Inputs/GVL_iXlinker.EtherCAT_Master_EPPxxxx.Beckhoff_EPP1xxx.Beckhoff_EPP1xxxEK1122.A_0018_EPP1321_0060_0016.A_0019_EPP1322_0001_0016.A_0020_EPP1322_0001_0017.A_0021_EPP1332_0001_0016.A_0022_EPP1332_0001_0017.A_0023_EPP1342_0001_0016.A_0024_EPP1342_0001_0017.A_0035_EPP1816_3008_0016.InfoData.AdsAddr <-> InfoData/AdsAddr
//     PlcTask Inputs/GVL_iXlinker.EtherCAT_Master_EPPxxxx.Beckhoff_EPP1xxx.Beckhoff_EPP1xxxEK1122.A_0018_EPP1321_0060_0016.A_0019_EPP1322_0001_0016.A_0020_EPP1322_0001_0017.A_0021_EPP1332_0001_0016.A_0022_EPP1332_0001_0017.A_0023_EPP1342_0001_0016.A_0024_EPP1342_0001_0017.A_0035_EPP1816_3008_0016.InfoData.State <-> InfoData/State
//   PLC/PLC Instance <-> EtherCAT Master EPPxxxx/Beckhoff EPP2xxx
//     PlcTask Inputs/GVL_iXlinker.EtherCAT_Master_EPPxxxx.Beckhoff_EPP2xxx.InfoData.State <-> InfoData/State
//   PLC/PLC Instance <-> EtherCAT Master EPPxxxx/Beckhoff EPP2xxx/Beckhoff EPP2xxxEK1122
//     PlcTask Inputs/GVL_iXlinker.EtherCAT_Master_EPPxxxx.Beckhoff_EPP2xxx.Beckhoff_EPP2xxxEK1122.InfoData.State <-> InfoData/State
//   PLC/PLC Instance <-> EtherCAT Master EPPxxxx/Beckhoff EPP2xxx/Beckhoff EPP2xxxEK1122/Beckhoff EPP2xxxsub EK1100
//     PlcTask Inputs/GVL_iXlinker.EtherCAT_Master_EPPxxxx.Beckhoff_EPP2xxx.Beckhoff_EPP2xxxEK1122.Beckhoff_EPP2xxxsub_EK1100.InfoData.State <-> InfoData/State
//   PLC/PLC Instance <-> EtherCAT Master EPPxxxx/Beckhoff EPP2xxx/Beckhoff EPP2xxxEK1122/A_0001(EPP2008-0001-0016)
//     PlcTask Outputs/GVL_iXlinker.EtherCAT_Master_EPPxxxx.Beckhoff_EPP2xxx.Beckhoff_EPP2xxxEK1122.A_0001_EPP2008_0001_0016.Channel_1.Output <-> Channel 1/Output
//     PlcTask Outputs/GVL_iXlinker.EtherCAT_Master_EPPxxxx.Beckhoff_EPP2xxx.Beckhoff_EPP2xxxEK1122.A_0001_EPP2008_0001_0016.Channel_2.Output <-> Channel 2/Output
//     PlcTask Outputs/GVL_iXlinker.EtherCAT_Master_EPPxxxx.Beckhoff_EPP2xxx.Beckhoff_EPP2xxxEK1122.A_0001_EPP2008_0001_0016.Channel_3.Output <-> Channel 3/Output
//     PlcTask Outputs/GVL_iXlinker.EtherCAT_Master_EPPxxxx.Beckhoff_EPP2xxx.Beckhoff_EPP2xxxEK1122.A_0001_EPP2008_0001_0016.Channel_4.Output <-> Channel 4/Output
//     PlcTask Outputs/GVL_iXlinker.EtherCAT_Master_EPPxxxx.Beckhoff_EPP2xxx.Beckhoff_EPP2xxxEK1122.A_0001_EPP2008_0001_0016.Channel_5.Output <-> Channel 5/Output
//     PlcTask Outputs/GVL_iXlinker.EtherCAT_Master_EPPxxxx.Beckhoff_EPP2xxx.Beckhoff_EPP2xxxEK1122.A_0001_EPP2008_0001_0016.Channel_6.Output <-> Channel 6/Output
//     PlcTask Outputs/GVL_iXlinker.EtherCAT_Master_EPPxxxx.Beckhoff_EPP2xxx.Beckhoff_EPP2xxxEK1122.A_0001_EPP2008_0001_0016.Channel_7.Output <-> Channel 7/Output
//     PlcTask Outputs/GVL_iXlinker.EtherCAT_Master_EPPxxxx.Beckhoff_EPP2xxx.Beckhoff_EPP2xxxEK1122.A_0001_EPP2008_0001_0016.Channel_8.Output <-> Channel 8/Output
//     PlcTask Inputs/GVL_iXlinker.EtherCAT_Master_EPPxxxx.Beckhoff_EPP2xxx.Beckhoff_EPP2xxxEK1122.A_0001_EPP2008_0001_0016.WcState.WcState <-> WcState/WcState
//     PlcTask Inputs/GVL_iXlinker.EtherCAT_Master_EPPxxxx.Beckhoff_EPP2xxx.Beckhoff_EPP2xxxEK1122.A_0001_EPP2008_0001_0016.InfoData.State <-> InfoData/State
//   PLC/PLC Instance <-> EtherCAT Master EPPxxxx/Beckhoff EPP2xxx/Beckhoff EPP2xxxEK1122/A_0002(EPP2008-0001-0017)
//     PlcTask Outputs/GVL_iXlinker.EtherCAT_Master_EPPxxxx.Beckhoff_EPP2xxx.Beckhoff_EPP2xxxEK1122.A_0002_EPP2008_0001_0017.Channel_1.Output <-> Channel 1/Output
//     PlcTask Outputs/GVL_iXlinker.EtherCAT_Master_EPPxxxx.Beckhoff_EPP2xxx.Beckhoff_EPP2xxxEK1122.A_0002_EPP2008_0001_0017.Channel_2.Output <-> Channel 2/Output
//     PlcTask Outputs/GVL_iXlinker.EtherCAT_Master_EPPxxxx.Beckhoff_EPP2xxx.Beckhoff_EPP2xxxEK1122.A_0002_EPP2008_0001_0017.Channel_3.Output <-> Channel 3/Output
//     PlcTask Outputs/GVL_iXlinker.EtherCAT_Master_EPPxxxx.Beckhoff_EPP2xxx.Beckhoff_EPP2xxxEK1122.A_0002_EPP2008_0001_0017.Channel_4.Output <-> Channel 4/Output
//     PlcTask Outputs/GVL_iXlinker.EtherCAT_Master_EPPxxxx.Beckhoff_EPP2xxx.Beckhoff_EPP2xxxEK1122.A_0002_EPP2008_0001_0017.Channel_5.Output <-> Channel 5/Output
//     PlcTask Outputs/GVL_iXlinker.EtherCAT_Master_EPPxxxx.Beckhoff_EPP2xxx.Beckhoff_EPP2xxxEK1122.A_0002_EPP2008_0001_0017.Channel_6.Output <-> Channel 6/Output
//     PlcTask Outputs/GVL_iXlinker.EtherCAT_Master_EPPxxxx.Beckhoff_EPP2xxx.Beckhoff_EPP2xxxEK1122.A_0002_EPP2008_0001_0017.Channel_7.Output <-> Channel 7/Output
//     PlcTask Outputs/GVL_iXlinker.EtherCAT_Master_EPPxxxx.Beckhoff_EPP2xxx.Beckhoff_EPP2xxxEK1122.A_0002_EPP2008_0001_0017.Channel_8.Output <-> Channel 8/Output
//     PlcTask Inputs/GVL_iXlinker.EtherCAT_Master_EPPxxxx.Beckhoff_EPP2xxx.Beckhoff_EPP2xxxEK1122.A_0002_EPP2008_0001_0017.WcState.WcState <-> WcState/WcState
//     PlcTask Inputs/GVL_iXlinker.EtherCAT_Master_EPPxxxx.Beckhoff_EPP2xxx.Beckhoff_EPP2xxxEK1122.A_0002_EPP2008_0001_0017.InfoData.State <-> InfoData/State
//   PLC/PLC Instance <-> EtherCAT Master EPPxxxx/Beckhoff EPP2xxx/Beckhoff EPP2xxxEK1122/A_0003(EPP2008-0001-0018)
//     PlcTask Outputs/GVL_iXlinker.EtherCAT_Master_EPPxxxx.Beckhoff_EPP2xxx.Beckhoff_EPP2xxxEK1122.A_0003_EPP2008_0001_0018.Channel_1.Output <-> Channel 1/Output
//     PlcTask Outputs/GVL_iXlinker.EtherCAT_Master_EPPxxxx.Beckhoff_EPP2xxx.Beckhoff_EPP2xxxEK1122.A_0003_EPP2008_0001_0018.Channel_2.Output <-> Channel 2/Output
//     PlcTask Outputs/GVL_iXlinker.EtherCAT_Master_EPPxxxx.Beckhoff_EPP2xxx.Beckhoff_EPP2xxxEK1122.A_0003_EPP2008_0001_0018.Channel_3.Output <-> Channel 3/Output
//     PlcTask Outputs/GVL_iXlinker.EtherCAT_Master_EPPxxxx.Beckhoff_EPP2xxx.Beckhoff_EPP2xxxEK1122.A_0003_EPP2008_0001_0018.Channel_4.Output <-> Channel 4/Output
//     PlcTask Outputs/GVL_iXlinker.EtherCAT_Master_EPPxxxx.Beckhoff_EPP2xxx.Beckhoff_EPP2xxxEK1122.A_0003_EPP2008_0001_0018.Channel_5.Output <-> Channel 5/Output
//     PlcTask Outputs/GVL_iXlinker.EtherCAT_Master_EPPxxxx.Beckhoff_EPP2xxx.Beckhoff_EPP2xxxEK1122.A_0003_EPP2008_0001_0018.Channel_6.Output <-> Channel 6/Output
//     PlcTask Outputs/GVL_iXlinker.EtherCAT_Master_EPPxxxx.Beckhoff_EPP2xxx.Beckhoff_EPP2xxxEK1122.A_0003_EPP2008_0001_0018.Channel_7.Output <-> Channel 7/Output
//     PlcTask Outputs/GVL_iXlinker.EtherCAT_Master_EPPxxxx.Beckhoff_EPP2xxx.Beckhoff_EPP2xxxEK1122.A_0003_EPP2008_0001_0018.Channel_8.Output <-> Channel 8/Output
//     PlcTask Inputs/GVL_iXlinker.EtherCAT_Master_EPPxxxx.Beckhoff_EPP2xxx.Beckhoff_EPP2xxxEK1122.A_0003_EPP2008_0001_0018.WcState.WcState <-> WcState/WcState
//     PlcTask Inputs/GVL_iXlinker.EtherCAT_Master_EPPxxxx.Beckhoff_EPP2xxx.Beckhoff_EPP2xxxEK1122.A_0003_EPP2008_0001_0018.InfoData.State <-> InfoData/State
//   PLC/PLC Instance <-> EtherCAT Master EPPxxxx/Beckhoff EPP2xxx/Beckhoff EPP2xxxEK1122/A_0004(EPP2008-0002-0016)
//     PlcTask Outputs/GVL_iXlinker.EtherCAT_Master_EPPxxxx.Beckhoff_EPP2xxx.Beckhoff_EPP2xxxEK1122.A_0004_EPP2008_0002_0016.Channel_1.Output <-> Channel 1/Output
//     PlcTask Outputs/GVL_iXlinker.EtherCAT_Master_EPPxxxx.Beckhoff_EPP2xxx.Beckhoff_EPP2xxxEK1122.A_0004_EPP2008_0002_0016.Channel_2.Output <-> Channel 2/Output
//     PlcTask Outputs/GVL_iXlinker.EtherCAT_Master_EPPxxxx.Beckhoff_EPP2xxx.Beckhoff_EPP2xxxEK1122.A_0004_EPP2008_0002_0016.Channel_3.Output <-> Channel 3/Output
//     PlcTask Outputs/GVL_iXlinker.EtherCAT_Master_EPPxxxx.Beckhoff_EPP2xxx.Beckhoff_EPP2xxxEK1122.A_0004_EPP2008_0002_0016.Channel_4.Output <-> Channel 4/Output
//     PlcTask Outputs/GVL_iXlinker.EtherCAT_Master_EPPxxxx.Beckhoff_EPP2xxx.Beckhoff_EPP2xxxEK1122.A_0004_EPP2008_0002_0016.Channel_5.Output <-> Channel 5/Output
//     PlcTask Outputs/GVL_iXlinker.EtherCAT_Master_EPPxxxx.Beckhoff_EPP2xxx.Beckhoff_EPP2xxxEK1122.A_0004_EPP2008_0002_0016.Channel_6.Output <-> Channel 6/Output
//     PlcTask Outputs/GVL_iXlinker.EtherCAT_Master_EPPxxxx.Beckhoff_EPP2xxx.Beckhoff_EPP2xxxEK1122.A_0004_EPP2008_0002_0016.Channel_7.Output <-> Channel 7/Output
//     PlcTask Outputs/GVL_iXlinker.EtherCAT_Master_EPPxxxx.Beckhoff_EPP2xxx.Beckhoff_EPP2xxxEK1122.A_0004_EPP2008_0002_0016.Channel_8.Output <-> Channel 8/Output
//     PlcTask Inputs/GVL_iXlinker.EtherCAT_Master_EPPxxxx.Beckhoff_EPP2xxx.Beckhoff_EPP2xxxEK1122.A_0004_EPP2008_0002_0016.WcState.WcState <-> WcState/WcState
//     PlcTask Inputs/GVL_iXlinker.EtherCAT_Master_EPPxxxx.Beckhoff_EPP2xxx.Beckhoff_EPP2xxxEK1122.A_0004_EPP2008_0002_0016.InfoData.State <-> InfoData/State
//   PLC/PLC Instance <-> EtherCAT Master EPPxxxx/Beckhoff EPP2xxx/Beckhoff EPP2xxxEK1122/A_0005(EPP2008-0002-0017)
//     PlcTask Outputs/GVL_iXlinker.EtherCAT_Master_EPPxxxx.Beckhoff_EPP2xxx.Beckhoff_EPP2xxxEK1122.A_0005_EPP2008_0002_0017.Channel_1.Output <-> Channel 1/Output
//     PlcTask Outputs/GVL_iXlinker.EtherCAT_Master_EPPxxxx.Beckhoff_EPP2xxx.Beckhoff_EPP2xxxEK1122.A_0005_EPP2008_0002_0017.Channel_2.Output <-> Channel 2/Output
//     PlcTask Outputs/GVL_iXlinker.EtherCAT_Master_EPPxxxx.Beckhoff_EPP2xxx.Beckhoff_EPP2xxxEK1122.A_0005_EPP2008_0002_0017.Channel_3.Output <-> Channel 3/Output
//     PlcTask Outputs/GVL_iXlinker.EtherCAT_Master_EPPxxxx.Beckhoff_EPP2xxx.Beckhoff_EPP2xxxEK1122.A_0005_EPP2008_0002_0017.Channel_4.Output <-> Channel 4/Output
//     PlcTask Outputs/GVL_iXlinker.EtherCAT_Master_EPPxxxx.Beckhoff_EPP2xxx.Beckhoff_EPP2xxxEK1122.A_0005_EPP2008_0002_0017.Channel_5.Output <-> Channel 5/Output
//     PlcTask Outputs/GVL_iXlinker.EtherCAT_Master_EPPxxxx.Beckhoff_EPP2xxx.Beckhoff_EPP2xxxEK1122.A_0005_EPP2008_0002_0017.Channel_6.Output <-> Channel 6/Output
//     PlcTask Outputs/GVL_iXlinker.EtherCAT_Master_EPPxxxx.Beckhoff_EPP2xxx.Beckhoff_EPP2xxxEK1122.A_0005_EPP2008_0002_0017.Channel_7.Output <-> Channel 7/Output
//     PlcTask Outputs/GVL_iXlinker.EtherCAT_Master_EPPxxxx.Beckhoff_EPP2xxx.Beckhoff_EPP2xxxEK1122.A_0005_EPP2008_0002_0017.Channel_8.Output <-> Channel 8/Output
//     PlcTask Inputs/GVL_iXlinker.EtherCAT_Master_EPPxxxx.Beckhoff_EPP2xxx.Beckhoff_EPP2xxxEK1122.A_0005_EPP2008_0002_0017.WcState.WcState <-> WcState/WcState
//     PlcTask Inputs/GVL_iXlinker.EtherCAT_Master_EPPxxxx.Beckhoff_EPP2xxx.Beckhoff_EPP2xxxEK1122.A_0005_EPP2008_0002_0017.InfoData.State <-> InfoData/State
//   PLC/PLC Instance <-> EtherCAT Master EPPxxxx/Beckhoff EPP2xxx/Beckhoff EPP2xxxEK1122/A_0006(EPP2008-0002-0018)
//     PlcTask Outputs/GVL_iXlinker.EtherCAT_Master_EPPxxxx.Beckhoff_EPP2xxx.Beckhoff_EPP2xxxEK1122.A_0006_EPP2008_0002_0018.Channel_1.Output <-> Channel 1/Output
//     PlcTask Outputs/GVL_iXlinker.EtherCAT_Master_EPPxxxx.Beckhoff_EPP2xxx.Beckhoff_EPP2xxxEK1122.A_0006_EPP2008_0002_0018.Channel_2.Output <-> Channel 2/Output
//     PlcTask Outputs/GVL_iXlinker.EtherCAT_Master_EPPxxxx.Beckhoff_EPP2xxx.Beckhoff_EPP2xxxEK1122.A_0006_EPP2008_0002_0018.Channel_3.Output <-> Channel 3/Output
//     PlcTask Outputs/GVL_iXlinker.EtherCAT_Master_EPPxxxx.Beckhoff_EPP2xxx.Beckhoff_EPP2xxxEK1122.A_0006_EPP2008_0002_0018.Channel_4.Output <-> Channel 4/Output
//     PlcTask Outputs/GVL_iXlinker.EtherCAT_Master_EPPxxxx.Beckhoff_EPP2xxx.Beckhoff_EPP2xxxEK1122.A_0006_EPP2008_0002_0018.Channel_5.Output <-> Channel 5/Output
//     PlcTask Outputs/GVL_iXlinker.EtherCAT_Master_EPPxxxx.Beckhoff_EPP2xxx.Beckhoff_EPP2xxxEK1122.A_0006_EPP2008_0002_0018.Channel_6.Output <-> Channel 6/Output
//     PlcTask Outputs/GVL_iXlinker.EtherCAT_Master_EPPxxxx.Beckhoff_EPP2xxx.Beckhoff_EPP2xxxEK1122.A_0006_EPP2008_0002_0018.Channel_7.Output <-> Channel 7/Output
//     PlcTask Outputs/GVL_iXlinker.EtherCAT_Master_EPPxxxx.Beckhoff_EPP2xxx.Beckhoff_EPP2xxxEK1122.A_0006_EPP2008_0002_0018.Channel_8.Output <-> Channel 8/Output
//     PlcTask Inputs/GVL_iXlinker.EtherCAT_Master_EPPxxxx.Beckhoff_EPP2xxx.Beckhoff_EPP2xxxEK1122.A_0006_EPP2008_0002_0018.WcState.WcState <-> WcState/WcState
//     PlcTask Inputs/GVL_iXlinker.EtherCAT_Master_EPPxxxx.Beckhoff_EPP2xxx.Beckhoff_EPP2xxxEK1122.A_0006_EPP2008_0002_0018.InfoData.State <-> InfoData/State
//   PLC/PLC Instance <-> EtherCAT Master EPPxxxx/Beckhoff EPP2xxx/Beckhoff EPP2xxxEK1122/A_0007(EPP2008-0022-0016)
//     PlcTask Outputs/GVL_iXlinker.EtherCAT_Master_EPPxxxx.Beckhoff_EPP2xxx.Beckhoff_EPP2xxxEK1122.A_0007_EPP2008_0022_0016.Channel_1.Output <-> Channel 1/Output
//     PlcTask Outputs/GVL_iXlinker.EtherCAT_Master_EPPxxxx.Beckhoff_EPP2xxx.Beckhoff_EPP2xxxEK1122.A_0007_EPP2008_0022_0016.Channel_2.Output <-> Channel 2/Output
//     PlcTask Outputs/GVL_iXlinker.EtherCAT_Master_EPPxxxx.Beckhoff_EPP2xxx.Beckhoff_EPP2xxxEK1122.A_0007_EPP2008_0022_0016.Channel_3.Output <-> Channel 3/Output
//     PlcTask Outputs/GVL_iXlinker.EtherCAT_Master_EPPxxxx.Beckhoff_EPP2xxx.Beckhoff_EPP2xxxEK1122.A_0007_EPP2008_0022_0016.Channel_4.Output <-> Channel 4/Output
//     PlcTask Outputs/GVL_iXlinker.EtherCAT_Master_EPPxxxx.Beckhoff_EPP2xxx.Beckhoff_EPP2xxxEK1122.A_0007_EPP2008_0022_0016.Channel_5.Output <-> Channel 5/Output
//     PlcTask Outputs/GVL_iXlinker.EtherCAT_Master_EPPxxxx.Beckhoff_EPP2xxx.Beckhoff_EPP2xxxEK1122.A_0007_EPP2008_0022_0016.Channel_6.Output <-> Channel 6/Output
//     PlcTask Outputs/GVL_iXlinker.EtherCAT_Master_EPPxxxx.Beckhoff_EPP2xxx.Beckhoff_EPP2xxxEK1122.A_0007_EPP2008_0022_0016.Channel_7.Output <-> Channel 7/Output
//     PlcTask Outputs/GVL_iXlinker.EtherCAT_Master_EPPxxxx.Beckhoff_EPP2xxx.Beckhoff_EPP2xxxEK1122.A_0007_EPP2008_0022_0016.Channel_8.Output <-> Channel 8/Output
//     PlcTask Inputs/GVL_iXlinker.EtherCAT_Master_EPPxxxx.Beckhoff_EPP2xxx.Beckhoff_EPP2xxxEK1122.A_0007_EPP2008_0022_0016.WcState.WcState <-> WcState/WcState
//     PlcTask Inputs/GVL_iXlinker.EtherCAT_Master_EPPxxxx.Beckhoff_EPP2xxx.Beckhoff_EPP2xxxEK1122.A_0007_EPP2008_0022_0016.InfoData.State <-> InfoData/State
//   PLC/PLC Instance <-> EtherCAT Master EPPxxxx/Beckhoff EPP2xxx/Beckhoff EPP2xxxEK1122/A_0008(EPP2028-0001-0016)
//     PlcTask Outputs/GVL_iXlinker.EtherCAT_Master_EPPxxxx.Beckhoff_EPP2xxx.Beckhoff_EPP2xxxEK1122.A_0008_EPP2028_0001_0016.Channel_1.Output <-> Channel 1/Output
//     PlcTask Outputs/GVL_iXlinker.EtherCAT_Master_EPPxxxx.Beckhoff_EPP2xxx.Beckhoff_EPP2xxxEK1122.A_0008_EPP2028_0001_0016.Channel_2.Output <-> Channel 2/Output
//     PlcTask Outputs/GVL_iXlinker.EtherCAT_Master_EPPxxxx.Beckhoff_EPP2xxx.Beckhoff_EPP2xxxEK1122.A_0008_EPP2028_0001_0016.Channel_3.Output <-> Channel 3/Output
//     PlcTask Outputs/GVL_iXlinker.EtherCAT_Master_EPPxxxx.Beckhoff_EPP2xxx.Beckhoff_EPP2xxxEK1122.A_0008_EPP2028_0001_0016.Channel_4.Output <-> Channel 4/Output
//     PlcTask Outputs/GVL_iXlinker.EtherCAT_Master_EPPxxxx.Beckhoff_EPP2xxx.Beckhoff_EPP2xxxEK1122.A_0008_EPP2028_0001_0016.Channel_5.Output <-> Channel 5/Output
//     PlcTask Outputs/GVL_iXlinker.EtherCAT_Master_EPPxxxx.Beckhoff_EPP2xxx.Beckhoff_EPP2xxxEK1122.A_0008_EPP2028_0001_0016.Channel_6.Output <-> Channel 6/Output
//     PlcTask Outputs/GVL_iXlinker.EtherCAT_Master_EPPxxxx.Beckhoff_EPP2xxx.Beckhoff_EPP2xxxEK1122.A_0008_EPP2028_0001_0016.Channel_7.Output <-> Channel 7/Output
//     PlcTask Outputs/GVL_iXlinker.EtherCAT_Master_EPPxxxx.Beckhoff_EPP2xxx.Beckhoff_EPP2xxxEK1122.A_0008_EPP2028_0001_0016.Channel_8.Output <-> Channel 8/Output
//     PlcTask Inputs/GVL_iXlinker.EtherCAT_Master_EPPxxxx.Beckhoff_EPP2xxx.Beckhoff_EPP2xxxEK1122.A_0008_EPP2028_0001_0016.WcState.WcState <-> WcState/WcState
//     PlcTask Inputs/GVL_iXlinker.EtherCAT_Master_EPPxxxx.Beckhoff_EPP2xxx.Beckhoff_EPP2xxxEK1122.A_0008_EPP2028_0001_0016.InfoData.State <-> InfoData/State
//   PLC/PLC Instance <-> EtherCAT Master EPPxxxx/Beckhoff EPP2xxx/Beckhoff EPP2xxxEK1122/A_0009(EPP2028-0001-0017)
//     PlcTask Outputs/GVL_iXlinker.EtherCAT_Master_EPPxxxx.Beckhoff_EPP2xxx.Beckhoff_EPP2xxxEK1122.A_0009_EPP2028_0001_0017.Channel_1.Output <-> Channel 1/Output
//     PlcTask Outputs/GVL_iXlinker.EtherCAT_Master_EPPxxxx.Beckhoff_EPP2xxx.Beckhoff_EPP2xxxEK1122.A_0009_EPP2028_0001_0017.Channel_2.Output <-> Channel 2/Output
//     PlcTask Outputs/GVL_iXlinker.EtherCAT_Master_EPPxxxx.Beckhoff_EPP2xxx.Beckhoff_EPP2xxxEK1122.A_0009_EPP2028_0001_0017.Channel_3.Output <-> Channel 3/Output
//     PlcTask Outputs/GVL_iXlinker.EtherCAT_Master_EPPxxxx.Beckhoff_EPP2xxx.Beckhoff_EPP2xxxEK1122.A_0009_EPP2028_0001_0017.Channel_4.Output <-> Channel 4/Output
//     PlcTask Outputs/GVL_iXlinker.EtherCAT_Master_EPPxxxx.Beckhoff_EPP2xxx.Beckhoff_EPP2xxxEK1122.A_0009_EPP2028_0001_0017.Channel_5.Output <-> Channel 5/Output
//     PlcTask Outputs/GVL_iXlinker.EtherCAT_Master_EPPxxxx.Beckhoff_EPP2xxx.Beckhoff_EPP2xxxEK1122.A_0009_EPP2028_0001_0017.Channel_6.Output <-> Channel 6/Output
//     PlcTask Outputs/GVL_iXlinker.EtherCAT_Master_EPPxxxx.Beckhoff_EPP2xxx.Beckhoff_EPP2xxxEK1122.A_0009_EPP2028_0001_0017.Channel_7.Output <-> Channel 7/Output
//     PlcTask Outputs/GVL_iXlinker.EtherCAT_Master_EPPxxxx.Beckhoff_EPP2xxx.Beckhoff_EPP2xxxEK1122.A_0009_EPP2028_0001_0017.Channel_8.Output <-> Channel 8/Output
//     PlcTask Inputs/GVL_iXlinker.EtherCAT_Master_EPPxxxx.Beckhoff_EPP2xxx.Beckhoff_EPP2xxxEK1122.A_0009_EPP2028_0001_0017.WcState.WcState <-> WcState/WcState
//     PlcTask Inputs/GVL_iXlinker.EtherCAT_Master_EPPxxxx.Beckhoff_EPP2xxx.Beckhoff_EPP2xxxEK1122.A_0009_EPP2028_0001_0017.InfoData.State <-> InfoData/State
//   PLC/PLC Instance <-> EtherCAT Master EPPxxxx/Beckhoff EPP2xxx/Beckhoff EPP2xxxEK1122/A_0010(EPP2028-0002-0016)
//     PlcTask Outputs/GVL_iXlinker.EtherCAT_Master_EPPxxxx.Beckhoff_EPP2xxx.Beckhoff_EPP2xxxEK1122.A_0010_EPP2028_0002_0016.Channel_1.Output <-> Channel 1/Output
//     PlcTask Outputs/GVL_iXlinker.EtherCAT_Master_EPPxxxx.Beckhoff_EPP2xxx.Beckhoff_EPP2xxxEK1122.A_0010_EPP2028_0002_0016.Channel_2.Output <-> Channel 2/Output
//     PlcTask Outputs/GVL_iXlinker.EtherCAT_Master_EPPxxxx.Beckhoff_EPP2xxx.Beckhoff_EPP2xxxEK1122.A_0010_EPP2028_0002_0016.Channel_3.Output <-> Channel 3/Output
//     PlcTask Outputs/GVL_iXlinker.EtherCAT_Master_EPPxxxx.Beckhoff_EPP2xxx.Beckhoff_EPP2xxxEK1122.A_0010_EPP2028_0002_0016.Channel_4.Output <-> Channel 4/Output
//     PlcTask Outputs/GVL_iXlinker.EtherCAT_Master_EPPxxxx.Beckhoff_EPP2xxx.Beckhoff_EPP2xxxEK1122.A_0010_EPP2028_0002_0016.Channel_5.Output <-> Channel 5/Output
//     PlcTask Outputs/GVL_iXlinker.EtherCAT_Master_EPPxxxx.Beckhoff_EPP2xxx.Beckhoff_EPP2xxxEK1122.A_0010_EPP2028_0002_0016.Channel_6.Output <-> Channel 6/Output
//     PlcTask Outputs/GVL_iXlinker.EtherCAT_Master_EPPxxxx.Beckhoff_EPP2xxx.Beckhoff_EPP2xxxEK1122.A_0010_EPP2028_0002_0016.Channel_7.Output <-> Channel 7/Output
//     PlcTask Outputs/GVL_iXlinker.EtherCAT_Master_EPPxxxx.Beckhoff_EPP2xxx.Beckhoff_EPP2xxxEK1122.A_0010_EPP2028_0002_0016.Channel_8.Output <-> Channel 8/Output
//     PlcTask Inputs/GVL_iXlinker.EtherCAT_Master_EPPxxxx.Beckhoff_EPP2xxx.Beckhoff_EPP2xxxEK1122.A_0010_EPP2028_0002_0016.WcState.WcState <-> WcState/WcState
//     PlcTask Inputs/GVL_iXlinker.EtherCAT_Master_EPPxxxx.Beckhoff_EPP2xxx.Beckhoff_EPP2xxxEK1122.A_0010_EPP2028_0002_0016.InfoData.State <-> InfoData/State
//   PLC/PLC Instance <-> EtherCAT Master EPPxxxx/Beckhoff EPP2xxx/Beckhoff EPP2xxxEK1122/A_0011(EPP2028-0002-0017)
//     PlcTask Outputs/GVL_iXlinker.EtherCAT_Master_EPPxxxx.Beckhoff_EPP2xxx.Beckhoff_EPP2xxxEK1122.A_0011_EPP2028_0002_0017.Channel_1.Output <-> Channel 1/Output
//     PlcTask Outputs/GVL_iXlinker.EtherCAT_Master_EPPxxxx.Beckhoff_EPP2xxx.Beckhoff_EPP2xxxEK1122.A_0011_EPP2028_0002_0017.Channel_2.Output <-> Channel 2/Output
//     PlcTask Outputs/GVL_iXlinker.EtherCAT_Master_EPPxxxx.Beckhoff_EPP2xxx.Beckhoff_EPP2xxxEK1122.A_0011_EPP2028_0002_0017.Channel_3.Output <-> Channel 3/Output
//     PlcTask Outputs/GVL_iXlinker.EtherCAT_Master_EPPxxxx.Beckhoff_EPP2xxx.Beckhoff_EPP2xxxEK1122.A_0011_EPP2028_0002_0017.Channel_4.Output <-> Channel 4/Output
//     PlcTask Outputs/GVL_iXlinker.EtherCAT_Master_EPPxxxx.Beckhoff_EPP2xxx.Beckhoff_EPP2xxxEK1122.A_0011_EPP2028_0002_0017.Channel_5.Output <-> Channel 5/Output
//     PlcTask Outputs/GVL_iXlinker.EtherCAT_Master_EPPxxxx.Beckhoff_EPP2xxx.Beckhoff_EPP2xxxEK1122.A_0011_EPP2028_0002_0017.Channel_6.Output <-> Channel 6/Output
//     PlcTask Outputs/GVL_iXlinker.EtherCAT_Master_EPPxxxx.Beckhoff_EPP2xxx.Beckhoff_EPP2xxxEK1122.A_0011_EPP2028_0002_0017.Channel_7.Output <-> Channel 7/Output
//     PlcTask Outputs/GVL_iXlinker.EtherCAT_Master_EPPxxxx.Beckhoff_EPP2xxx.Beckhoff_EPP2xxxEK1122.A_0011_EPP2028_0002_0017.Channel_8.Output <-> Channel 8/Output
//     PlcTask Inputs/GVL_iXlinker.EtherCAT_Master_EPPxxxx.Beckhoff_EPP2xxx.Beckhoff_EPP2xxxEK1122.A_0011_EPP2028_0002_0017.WcState.WcState <-> WcState/WcState
//     PlcTask Inputs/GVL_iXlinker.EtherCAT_Master_EPPxxxx.Beckhoff_EPP2xxx.Beckhoff_EPP2xxxEK1122.A_0011_EPP2028_0002_0017.InfoData.State <-> InfoData/State
//   PLC/PLC Instance <-> EtherCAT Master EPPxxxx/Beckhoff EPP2xxx/Beckhoff EPP2xxxEK1122/A_0012(EPP2038-0001-0016)
//     PlcTask Inputs/GVL_iXlinker.EtherCAT_Master_EPPxxxx.Beckhoff_EPP2xxx.Beckhoff_EPP2xxxEK1122.A_0012_EPP2038_0001_0016.Diag_Channel_1.Input <-> Diag Channel 1/Input
//     PlcTask Inputs/GVL_iXlinker.EtherCAT_Master_EPPxxxx.Beckhoff_EPP2xxx.Beckhoff_EPP2xxxEK1122.A_0012_EPP2038_0001_0016.Diag_Channel_2.Input <-> Diag Channel 2/Input
//     PlcTask Inputs/GVL_iXlinker.EtherCAT_Master_EPPxxxx.Beckhoff_EPP2xxx.Beckhoff_EPP2xxxEK1122.A_0012_EPP2038_0001_0016.Diag_Channel_3.Input <-> Diag Channel 3/Input
//     PlcTask Inputs/GVL_iXlinker.EtherCAT_Master_EPPxxxx.Beckhoff_EPP2xxx.Beckhoff_EPP2xxxEK1122.A_0012_EPP2038_0001_0016.Diag_Channel_4.Input <-> Diag Channel 4/Input
//     PlcTask Inputs/GVL_iXlinker.EtherCAT_Master_EPPxxxx.Beckhoff_EPP2xxx.Beckhoff_EPP2xxxEK1122.A_0012_EPP2038_0001_0016.Diag_Channel_5.Input <-> Diag Channel 5/Input
//     PlcTask Inputs/GVL_iXlinker.EtherCAT_Master_EPPxxxx.Beckhoff_EPP2xxx.Beckhoff_EPP2xxxEK1122.A_0012_EPP2038_0001_0016.Diag_Channel_6.Input <-> Diag Channel 6/Input
//     PlcTask Inputs/GVL_iXlinker.EtherCAT_Master_EPPxxxx.Beckhoff_EPP2xxx.Beckhoff_EPP2xxxEK1122.A_0012_EPP2038_0001_0016.Diag_Channel_7.Input <-> Diag Channel 7/Input
//     PlcTask Inputs/GVL_iXlinker.EtherCAT_Master_EPPxxxx.Beckhoff_EPP2xxx.Beckhoff_EPP2xxxEK1122.A_0012_EPP2038_0001_0016.Diag_Channel_8.Input <-> Diag Channel 8/Input
//     PlcTask Outputs/GVL_iXlinker.EtherCAT_Master_EPPxxxx.Beckhoff_EPP2xxx.Beckhoff_EPP2xxxEK1122.A_0012_EPP2038_0001_0016.Channel_1.Output <-> Channel 1/Output
//     PlcTask Outputs/GVL_iXlinker.EtherCAT_Master_EPPxxxx.Beckhoff_EPP2xxx.Beckhoff_EPP2xxxEK1122.A_0012_EPP2038_0001_0016.Channel_2.Output <-> Channel 2/Output
//     PlcTask Outputs/GVL_iXlinker.EtherCAT_Master_EPPxxxx.Beckhoff_EPP2xxx.Beckhoff_EPP2xxxEK1122.A_0012_EPP2038_0001_0016.Channel_3.Output <-> Channel 3/Output
//     PlcTask Outputs/GVL_iXlinker.EtherCAT_Master_EPPxxxx.Beckhoff_EPP2xxx.Beckhoff_EPP2xxxEK1122.A_0012_EPP2038_0001_0016.Channel_4.Output <-> Channel 4/Output
//     PlcTask Outputs/GVL_iXlinker.EtherCAT_Master_EPPxxxx.Beckhoff_EPP2xxx.Beckhoff_EPP2xxxEK1122.A_0012_EPP2038_0001_0016.Channel_5.Output <-> Channel 5/Output
//     PlcTask Outputs/GVL_iXlinker.EtherCAT_Master_EPPxxxx.Beckhoff_EPP2xxx.Beckhoff_EPP2xxxEK1122.A_0012_EPP2038_0001_0016.Channel_6.Output <-> Channel 6/Output
//     PlcTask Outputs/GVL_iXlinker.EtherCAT_Master_EPPxxxx.Beckhoff_EPP2xxx.Beckhoff_EPP2xxxEK1122.A_0012_EPP2038_0001_0016.Channel_7.Output <-> Channel 7/Output
//     PlcTask Outputs/GVL_iXlinker.EtherCAT_Master_EPPxxxx.Beckhoff_EPP2xxx.Beckhoff_EPP2xxxEK1122.A_0012_EPP2038_0001_0016.Channel_8.Output <-> Channel 8/Output
//     PlcTask Inputs/GVL_iXlinker.EtherCAT_Master_EPPxxxx.Beckhoff_EPP2xxx.Beckhoff_EPP2xxxEK1122.A_0012_EPP2038_0001_0016.WcState.WcState <-> WcState/WcState
//     PlcTask Inputs/GVL_iXlinker.EtherCAT_Master_EPPxxxx.Beckhoff_EPP2xxx.Beckhoff_EPP2xxxEK1122.A_0012_EPP2038_0001_0016.WcState.InputToggle <-> WcState/InputToggle
//     PlcTask Inputs/GVL_iXlinker.EtherCAT_Master_EPPxxxx.Beckhoff_EPP2xxx.Beckhoff_EPP2xxxEK1122.A_0012_EPP2038_0001_0016.InfoData.State <-> InfoData/State
//   PLC/PLC Instance <-> EtherCAT Master EPPxxxx/Beckhoff EPP2xxx/Beckhoff EPP2xxxEK1122/A_0013(EPP2038-0002-0016)
//     PlcTask Inputs/GVL_iXlinker.EtherCAT_Master_EPPxxxx.Beckhoff_EPP2xxx.Beckhoff_EPP2xxxEK1122.A_0013_EPP2038_0002_0016.Diag_Channel_1.Input <-> Diag Channel 1/Input
//     PlcTask Inputs/GVL_iXlinker.EtherCAT_Master_EPPxxxx.Beckhoff_EPP2xxx.Beckhoff_EPP2xxxEK1122.A_0013_EPP2038_0002_0016.Diag_Channel_2.Input <-> Diag Channel 2/Input
//     PlcTask Inputs/GVL_iXlinker.EtherCAT_Master_EPPxxxx.Beckhoff_EPP2xxx.Beckhoff_EPP2xxxEK1122.A_0013_EPP2038_0002_0016.Diag_Channel_3.Input <-> Diag Channel 3/Input
//     PlcTask Inputs/GVL_iXlinker.EtherCAT_Master_EPPxxxx.Beckhoff_EPP2xxx.Beckhoff_EPP2xxxEK1122.A_0013_EPP2038_0002_0016.Diag_Channel_4.Input <-> Diag Channel 4/Input
//     PlcTask Inputs/GVL_iXlinker.EtherCAT_Master_EPPxxxx.Beckhoff_EPP2xxx.Beckhoff_EPP2xxxEK1122.A_0013_EPP2038_0002_0016.Diag_Channel_5.Input <-> Diag Channel 5/Input
//     PlcTask Inputs/GVL_iXlinker.EtherCAT_Master_EPPxxxx.Beckhoff_EPP2xxx.Beckhoff_EPP2xxxEK1122.A_0013_EPP2038_0002_0016.Diag_Channel_6.Input <-> Diag Channel 6/Input
//     PlcTask Inputs/GVL_iXlinker.EtherCAT_Master_EPPxxxx.Beckhoff_EPP2xxx.Beckhoff_EPP2xxxEK1122.A_0013_EPP2038_0002_0016.Diag_Channel_7.Input <-> Diag Channel 7/Input
//     PlcTask Inputs/GVL_iXlinker.EtherCAT_Master_EPPxxxx.Beckhoff_EPP2xxx.Beckhoff_EPP2xxxEK1122.A_0013_EPP2038_0002_0016.Diag_Channel_8.Input <-> Diag Channel 8/Input
//     PlcTask Outputs/GVL_iXlinker.EtherCAT_Master_EPPxxxx.Beckhoff_EPP2xxx.Beckhoff_EPP2xxxEK1122.A_0013_EPP2038_0002_0016.Channel_1.Output <-> Channel 1/Output
//     PlcTask Outputs/GVL_iXlinker.EtherCAT_Master_EPPxxxx.Beckhoff_EPP2xxx.Beckhoff_EPP2xxxEK1122.A_0013_EPP2038_0002_0016.Channel_2.Output <-> Channel 2/Output
//     PlcTask Outputs/GVL_iXlinker.EtherCAT_Master_EPPxxxx.Beckhoff_EPP2xxx.Beckhoff_EPP2xxxEK1122.A_0013_EPP2038_0002_0016.Channel_3.Output <-> Channel 3/Output
//     PlcTask Outputs/GVL_iXlinker.EtherCAT_Master_EPPxxxx.Beckhoff_EPP2xxx.Beckhoff_EPP2xxxEK1122.A_0013_EPP2038_0002_0016.Channel_4.Output <-> Channel 4/Output
//     PlcTask Outputs/GVL_iXlinker.EtherCAT_Master_EPPxxxx.Beckhoff_EPP2xxx.Beckhoff_EPP2xxxEK1122.A_0013_EPP2038_0002_0016.Channel_5.Output <-> Channel 5/Output
//     PlcTask Outputs/GVL_iXlinker.EtherCAT_Master_EPPxxxx.Beckhoff_EPP2xxx.Beckhoff_EPP2xxxEK1122.A_0013_EPP2038_0002_0016.Channel_6.Output <-> Channel 6/Output
//     PlcTask Outputs/GVL_iXlinker.EtherCAT_Master_EPPxxxx.Beckhoff_EPP2xxx.Beckhoff_EPP2xxxEK1122.A_0013_EPP2038_0002_0016.Channel_7.Output <-> Channel 7/Output
//     PlcTask Outputs/GVL_iXlinker.EtherCAT_Master_EPPxxxx.Beckhoff_EPP2xxx.Beckhoff_EPP2xxxEK1122.A_0013_EPP2038_0002_0016.Channel_8.Output <-> Channel 8/Output
//     PlcTask Inputs/GVL_iXlinker.EtherCAT_Master_EPPxxxx.Beckhoff_EPP2xxx.Beckhoff_EPP2xxxEK1122.A_0013_EPP2038_0002_0016.WcState.WcState <-> WcState/WcState
//     PlcTask Inputs/GVL_iXlinker.EtherCAT_Master_EPPxxxx.Beckhoff_EPP2xxx.Beckhoff_EPP2xxxEK1122.A_0013_EPP2038_0002_0016.WcState.InputToggle <-> WcState/InputToggle
//     PlcTask Inputs/GVL_iXlinker.EtherCAT_Master_EPPxxxx.Beckhoff_EPP2xxx.Beckhoff_EPP2xxxEK1122.A_0013_EPP2038_0002_0016.InfoData.State <-> InfoData/State
//   PLC/PLC Instance <-> EtherCAT Master EPPxxxx/Beckhoff EPP2xxx/Beckhoff EPP2xxxEK1122/A_0014(EPP2304-0061-0016)
//     PlcTask Inputs/GVL_iXlinker.EtherCAT_Master_EPPxxxx.Beckhoff_EPP2xxx.Beckhoff_EPP2xxxEK1122.A_0014_EPP2304_0061_0016.Channel_1.Input <-> Channel 1/Input
//     PlcTask Inputs/GVL_iXlinker.EtherCAT_Master_EPPxxxx.Beckhoff_EPP2xxx.Beckhoff_EPP2xxxEK1122.A_0014_EPP2304_0061_0016.Channel_2.Input <-> Channel 2/Input
//     PlcTask Outputs/GVL_iXlinker.EtherCAT_Master_EPPxxxx.Beckhoff_EPP2xxx.Beckhoff_EPP2xxxEK1122.A_0014_EPP2304_0061_0016.Channel_3.Output <-> Channel 3/Output
//     PlcTask Outputs/GVL_iXlinker.EtherCAT_Master_EPPxxxx.Beckhoff_EPP2xxx.Beckhoff_EPP2xxxEK1122.A_0014_EPP2304_0061_0016.Channel_4.Output <-> Channel 4/Output
//     PlcTask Inputs/GVL_iXlinker.EtherCAT_Master_EPPxxxx.Beckhoff_EPP2xxx.Beckhoff_EPP2xxxEK1122.A_0014_EPP2304_0061_0016.WcState.WcState <-> WcState/WcState
//     PlcTask Inputs/GVL_iXlinker.EtherCAT_Master_EPPxxxx.Beckhoff_EPP2xxx.Beckhoff_EPP2xxxEK1122.A_0014_EPP2304_0061_0016.WcState.InputToggle <-> WcState/InputToggle
//     PlcTask Inputs/GVL_iXlinker.EtherCAT_Master_EPPxxxx.Beckhoff_EPP2xxx.Beckhoff_EPP2xxxEK1122.A_0014_EPP2304_0061_0016.InfoData.State <-> InfoData/State
//   PLC/PLC Instance <-> EtherCAT Master EPPxxxx/Beckhoff EPP2xxx/Beckhoff EPP2xxxEK1122/A_0015(EPP2304-0061-0017)
//     PlcTask Inputs/GVL_iXlinker.EtherCAT_Master_EPPxxxx.Beckhoff_EPP2xxx.Beckhoff_EPP2xxxEK1122.A_0015_EPP2304_0061_0017.Channel_1.Input <-> Channel 1/Input
//     PlcTask Inputs/GVL_iXlinker.EtherCAT_Master_EPPxxxx.Beckhoff_EPP2xxx.Beckhoff_EPP2xxxEK1122.A_0015_EPP2304_0061_0017.Channel_2.Input <-> Channel 2/Input
//     PlcTask Outputs/GVL_iXlinker.EtherCAT_Master_EPPxxxx.Beckhoff_EPP2xxx.Beckhoff_EPP2xxxEK1122.A_0015_EPP2304_0061_0017.Channel_3.Output <-> Channel 3/Output
//     PlcTask Outputs/GVL_iXlinker.EtherCAT_Master_EPPxxxx.Beckhoff_EPP2xxx.Beckhoff_EPP2xxxEK1122.A_0015_EPP2304_0061_0017.Channel_4.Output <-> Channel 4/Output
//     PlcTask Inputs/GVL_iXlinker.EtherCAT_Master_EPPxxxx.Beckhoff_EPP2xxx.Beckhoff_EPP2xxxEK1122.A_0015_EPP2304_0061_0017.WcState.WcState <-> WcState/WcState
//     PlcTask Inputs/GVL_iXlinker.EtherCAT_Master_EPPxxxx.Beckhoff_EPP2xxx.Beckhoff_EPP2xxxEK1122.A_0015_EPP2304_0061_0017.WcState.InputToggle <-> WcState/InputToggle
//     PlcTask Inputs/GVL_iXlinker.EtherCAT_Master_EPPxxxx.Beckhoff_EPP2xxx.Beckhoff_EPP2xxxEK1122.A_0015_EPP2304_0061_0017.InfoData.State <-> InfoData/State
//   PLC/PLC Instance <-> EtherCAT Master EPPxxxx/Beckhoff EPP2xxx/Beckhoff EPP2xxxEK1122/A_0016(EPP2304-0061-0018)
//     PlcTask Inputs/GVL_iXlinker.EtherCAT_Master_EPPxxxx.Beckhoff_EPP2xxx.Beckhoff_EPP2xxxEK1122.A_0016_EPP2304_0061_0018.Channel_1.Input <-> Channel 1/Input
